C03638=1029.081,200.605,387.413,169.449,45.503,158.607
C03639=1029.086,200.854,387.389,169.452,45.500,158.607
C03640=1029.092,201.102,387.364,169.456,45.498,158.607
C03641=1029.098,201.351,387.340,169.460,45.496,158.607
C03642=1029.104,201.600,387.315,169.464,45.494,158.607
C03643=1029.110,201.849,387.290,169.468,45.491,158.607
C03644=1029.116,202.097,387.266,169.471,45.488,158.607
C03645=1029.122,202.346,387.240,169.474,45.486,158.607
C03646=1029.128,202.595,387.216,169.479,45.484,158.607
C03647=1029.134,202.843,387.191,169.482,45.482,158.607
C03648=1029.140,203.092,387.167,169.486,45.479,158.607
C03649=1029.146,203.341,387.142,169.490,45.477,158.606
C03650=1029.151,203.589,387.117,169.494,45.475,158.606
C03651=1029.157,203.839,387.092,169.498,45.472,158.606
C03652=1029.182,204.885,386.988,169.864,45.576,158.667
C03653=1029.194,205.258,386.949,169.867,45.574,158.667
C03654=1029.203,205.632,386.909,169.872,45.571,158.667
C03655=1029.213,206.005,386.870,169.876,45.569,158.667
C03656=1029.223,206.378,386.831,169.880,45.566,158.667
C03657=1029.230,206.628,386.805,169.883,45.565,158.667
C03658=1029.236,206.876,386.779,169.886,45.564,158.667
C03659=1029.243,207.124,386.752,169.889,45.562,158.667
C03660=1029.250,207.372,386.726,169.892,45.560,158.667
C03661=1029.256,207.621,386.699,169.895,45.559,158.667
C03662=1029.263,207.870,386.673,169.897,45.557,158.667
C03663=1029.270,208.118,386.647,169.900,45.556,158.667
C03664=1029.277,208.367,386.620,169.903,45.554,158.667
C03665=1029.284,208.615,386.594,169.905,45.553,158.667
C03666=1029.290,208.864,386.567,169.908,45.551,158.667
C03667=1029.297,209.112,386.541,169.911,45.550,158.667
C03668=1029.304,209.361,386.515,169.914,45.549,158.667
C03669=1029.309,209.609,386.488,169.916,45.547,158.666
C03670=1029.317,209.858,386.462,169.919,45.545,158.666
C03671=1029.324,210.107,386.435,169.923,45.544,158.666
C03672=1029.330,210.355,386.409,169.926,45.542,158.666
C03673=1029.337,210.604,386.382,169.928,45.541,158.667
C03674=1029.343,210.852,386.356,169.931,45.540,158.667
C03675=1029.350,211.101,386.330,169.934,45.538,158.666
C03676=1029.356,211.349,386.303,169.936,45.536,158.666
C03677=1029.363,211.598,386.277,169.939,45.535,158.666
C03678=1029.370,211.846,386.249,169.942,45.534,158.666
C03679=1029.376,212.094,386.223,169.945,45.532,158.666
C03680=1029.383,212.343,386.196,169.948,45.531,158.666
C03681=1029.389,212.591,386.170,169.950,45.530,158.666
C03682=1029.396,212.840,386.144,169.954,45.528,158.666
C03683=1029.403,213.089,386.117,169.957,45.527,158.667
C03684=1029.409,213.337,386.090,169.960,45.525,158.667
C03685=1029.416,213.586,386.063,169.962,45.524,158.667
C03686=1029.422,213.834,386.037,169.965,45.523,158.667
C03687=1029.429,214.083,386.010,169.968,45.521,158.667
C03688=1029.436,214.331,385.983,169.970,45.519,158.666
C03689=1029.442,214.579,385.956,169.973,45.518,158.666
C03690=1029.449,214.828,385.929,169.976,45.517,158.666
C03691=1029.456,215.077,385.903,169.979,45.515,158.666
C03692=1029.462,215.325,385.876,169.983,45.514,158.666
C03693=1029.469,215.573,385.849,169.985,45.512,158.666
C03694=1029.476,215.822,385.822,169.988,45.511,158.667
C03695=1029.482,216.070,385.796,169.991,45.510,158.667
C03696=1029.489,216.319,385.768,169.994,45.508,158.667
C03697=1029.496,216.568,385.742,169.996,45.507,158.667
C03698=1029.502,216.816,385.715,169.999,45.506,158.667
C03699=1029.509,217.064,385.688,170.002,45.504,158.667
C03700=1029.516,217.313,385.661,170.006,45.503,158.667
C03701=1029.523,217.562,385.635,170.009,45.501,158.667
C03702=1029.529,217.810,385.607,170.011,45.500,158.667
C03703=1029.536,218.058,385.581,170.014,45.499,158.667
C03704=1029.543,218.307,385.553,170.017,45.497,158.667
C03705=1029.549,218.555,385.527,170.020,45.496,158.667
C03706=1029.556,218.804,385.501,170.023,45.495,158.667
C03707=1029.563,219.052,385.473,170.026,45.493,158.667
C03708=1029.570,219.301,385.447,170.029,45.492,158.667
C03709=1029.579,219.679,385.406,170.034,45.490,158.667
C03710=1029.589,220.058,385.364,170.037,45.488,158.667
C03711=1029.599,220.437,385.322,170.042,45.486,158.667
C03712=1029.609,220.816,385.281,170.047,45.484,158.667
C03713=1029.616,221.065,385.254,170.050,45.483,158.667
C03714=1029.623,221.313,385.227,170.052,45.482,158.667
C03715=1029.630,221.562,385.200,170.055,45.480,158.667
C03716=1029.636,221.810,385.172,170.058,45.479,158.667
C03717=1029.642,222.059,385.145,170.062,45.477,158.667
C03718=1029.649,222.307,385.118,170.064,45.476,158.667
C03719=1029.656,222.556,385.090,170.068,45.475,158.667
C03720=1029.662,222.804,385.064,170.070,45.474,158.667
C03721=1029.669,223.053,385.036,170.073,45.473,158.667
C03722=1029.676,223.301,385.009,170.076,45.471,158.667
C03723=1029.682,223.550,384.982,170.079,45.470,158.667
C03724=1029.689,223.798,384.954,170.082,45.468,158.667
C03725=1029.695,224.046,384.927,170.085,45.467,158.667
C03726=1029.701,224.295,384.900,170.088,45.466,158.668
C03727=1029.709,224.543,384.873,170.091,45.465,158.668
C03728=1029.716,224.792,384.845,170.094,45.464,158.668
C03729=1029.722,225.041,384.818,170.098,45.462,158.668
C03730=1029.729,225.289,384.790,170.100,45.461,158.668
C03731=1029.735,225.537,384.763,170.103,45.460,158.668
C03732=1029.742,225.785,384.736,170.106,45.459,158.668
C03733=1029.749,226.034,384.709,170.109,45.457,158.668
C03734=1029.755,226.282,384.681,170.112,45.456,158.668
C03735=1029.763,226.531,384.654,170.115,45.454,158.668
C03736=1029.769,226.779,384.626,170.118,45.454,158.668
C03737=1029.776,227.027,384.598,170.121,45.452,158.668
C03738=1029.782,227.276,384.572,170.124,45.451,158.668
C03739=1029.789,227.524,384.545,170.127,45.450,158.668
C03740=1029.796,227.772,384.517,170.131,45.448,158.668
C03741=1029.803,228.021,384.489,170.134,45.447,158.668
C03742=1029.809,228.269,384.461,170.136,45.446,158.668
C03743=1029.816,228.518,384.434,170.139,45.445,158.668
C03744=1029.823,228.766,384.406,170.142,45.444,158.669
C03745=1029.829,229.015,384.378,170.146,45.443,158.669
C03746=1029.835,229.262,384.351,170.149,45.441,158.669
C03747=1029.842,229.511,384.324,170.152,45.440,158.669
C03748=1029.848,229.760,384.296,170.155,45.439,158.669
C03749=1029.855,230.008,384.268,170.157,45.438,158.669
C03750=1029.862,230.257,384.241,170.161,45.437,158.669
C03751=1029.868,230.505,384.213,170.164,45.436,158.669
C03752=1029.875,230.754,384.185,170.167,45.434,158.669
C03753=1029.882,231.002,384.157,170.170,45.433,158.669
C03754=1029.888,231.250,384.130,170.173,45.432,158.669
C03755=1029.895,231.499,384.101,170.176,45.431,158.669
C03756=1029.901,231.747,384.073,170.180,45.430,158.669
C03757=1029.908,231.995,384.045,170.182,45.429,158.669
C03758=1029.914,232.243,384.018,170.185,45.428,158.670
C03759=1029.921,232.492,383.990,170.188,45.427,158.670
C03760=1029.928,232.740,383.962,170.191,45.426,158.670
C03761=1029.933,232.989,383.934,170.195,45.424,158.670
C03762=1029.940,233.237,383.906,170.198,45.424,158.670
C03763=1029.947,233.485,383.878,170.201,45.422,158.670
C03764=1029.954,233.734,383.850,170.204,45.422,158.670
C03765=1029.964,234.105,383.808,170.209,45.420,158.670
C03766=1029.973,234.476,383.766,170.213,45.418,158.670
C03767=1029.984,234.848,383.725,170.218,45.416,158.671
C03768=1029.994,235.219,383.683,170.223,45.414,158.671
C03769=1030.000,235.467,383.655,170.226,45.414,158.671
C03770=1030.006,235.716,383.627,170.229,45.412,158.671
C03771=1030.013,235.964,383.599,170.232,45.412,158.671
C03772=1030.020,236.212,383.571,170.236,45.410,158.671
C03773=1030.026,236.460,383.543,170.239,45.409,158.671
C03774=1030.033,236.709,383.515,170.241,45.408,158.671
C03775=1030.040,236.958,383.487,170.244,45.407,158.671
C03776=1030.047,237.206,383.458,170.248,45.406,158.671
C03777=1030.053,237.455,383.430,170.251,45.405,158.672
C03778=1030.060,237.703,383.403,170.254,45.404,158.672
C03779=1030.067,237.951,383.374,170.257,45.403,158.672
C03780=1030.073,238.200,383.346,170.261,45.401,158.672
C03781=1030.080,238.448,383.318,170.264,45.401,158.672
C03782=1030.087,238.696,383.290,170.267,45.400,158.672
C03783=1030.093,238.944,383.262,170.270,45.399,158.672
C03784=1030.100,239.192,383.233,170.274,45.398,158.672
C03785=1030.106,239.441,383.205,170.277,45.396,158.672
C03786=1030.113,239.689,383.177,170.280,45.396,158.673
C03787=1030.120,239.937,383.149,170.282,45.394,158.673
C03788=1030.126,240.187,383.120,170.286,45.394,158.673
C03789=1030.133,240.434,383.092,170.289,45.393,158.673
C03790=1030.139,240.683,383.064,170.292,45.392,158.673
C03791=1030.146,240.931,383.035,170.295,45.391,158.673
C03792=1030.153,241.179,383.007,170.299,45.390,158.673
C03793=1030.159,241.428,382.978,170.302,45.389,158.673
C03794=1030.166,241.675,382.950,170.305,45.388,158.674
C03795=1030.172,241.924,382.922,170.309,45.387,158.674
C03796=1030.179,242.172,382.893,170.312,45.386,158.674
C03797=1030.186,242.421,382.864,170.315,45.385,158.674
C03798=1030.193,242.669,382.836,170.318,45.384,158.674
C03799=1030.199,242.917,382.807,170.322,45.383,158.674
C03800=1030.206,243.165,382.778,170.325,45.382,158.674
C03801=1030.212,243.414,382.750,170.328,45.381,158.675
C03802=1030.219,243.662,382.722,170.331,45.381,158.675
C03803=1030.225,243.910,382.693,170.335,45.380,158.675
C03804=1030.232,244.159,382.665,170.338,45.378,158.675
C03805=1030.239,244.407,382.636,170.341,45.378,158.675
C03806=1030.245,244.655,382.606,170.345,45.377,158.675
C03807=1030.251,244.903,382.577,170.348,45.376,158.675
C03808=1030.258,245.152,382.550,170.351,45.375,158.676
C03809=1030.264,245.400,382.521,170.354,45.375,158.676
C03810=1030.270,245.648,382.492,170.358,45.373,158.676
C03811=1030.277,245.897,382.462,170.361,45.372,158.676
C03812=1030.284,246.145,382.434,170.364,45.372,158.676
C03813=1030.290,246.393,382.405,170.367,45.371,158.676
C03814=1030.297,246.641,382.376,170.371,45.370,158.677
C03815=1030.303,246.890,382.347,170.374,45.369,158.677
C03816=1030.310,247.138,382.319,170.377,45.369,158.677
C03817=1030.317,247.386,382.290,170.380,45.368,158.677
C03818=1030.323,247.635,382.260,170.384,45.367,158.677
C03819=1030.329,247.883,382.231,170.387,45.366,158.677
C03820=1030.335,248.131,382.202,170.390,45.365,158.678
C03821=1030.346,248.497,382.160,170.395,45.364,158.678
C03822=1030.355,248.861,382.117,170.400,45.363,158.678
C03823=1030.365,249.227,382.074,170.405,45.362,158.678
C03824=1030.374,249.592,382.032,170.410,45.360,158.679
C03825=1030.381,249.840,382.003,170.413,45.360,158.679
C03826=1030.387,250.089,381.973,170.416,45.359,158.679
C03827=1030.394,250.337,381.945,170.420,45.358,158.679
C03828=1030.401,250.585,381.916,170.423,45.357,158.679
C03829=1030.407,250.834,381.887,170.426,45.357,158.680
C03830=1030.414,251.082,381.858,170.430,45.356,158.680
C03831=1030.420,251.330,381.828,170.433,45.355,158.680
C03832=1030.427,251.577,381.799,170.436,45.354,158.680
C03833=1030.434,251.826,381.770,170.440,45.353,158.680
C03834=1030.440,252.074,381.741,170.443,45.353,158.680
C03835=1030.447,252.323,381.712,170.446,45.352,158.681
C03836=1030.453,252.571,381.682,170.451,45.351,158.681
C03837=1030.460,252.819,381.654,170.454,45.350,158.681
C03838=1030.467,253.067,381.625,170.457,45.349,158.681
C03839=1030.474,253.316,381.595,170.461,45.349,158.681
C03840=1030.480,253.564,381.566,170.464,45.348,158.682
C03841=1030.487,253.813,381.536,170.468,45.347,158.682
C03842=1030.494,254.060,381.508,170.471,45.347,158.682
C03843=1030.500,254.308,381.479,170.474,45.346,158.682
C03844=1030.507,254.557,381.449,170.478,45.345,158.682
C03845=1030.514,254.805,381.420,170.481,45.344,158.682
C03846=1030.520,255.054,381.390,170.485,45.343,158.683
C03847=1030.527,255.301,381.362,170.488,45.343,158.683
C03848=1030.534,255.549,381.332,170.491,45.342,158.683
C03849=1030.541,255.798,381.303,170.495,45.341,158.683
C03850=1030.547,256.046,381.274,170.498,45.340,158.683
C03851=1030.554,256.294,381.244,170.502,45.339,158.684
C03852=1030.560,256.542,381.215,170.505,45.339,158.684
C03853=1030.568,256.791,381.186,170.508,45.338,158.684
C03854=1030.575,257.038,381.156,170.512,45.337,158.684
C03855=1030.581,257.287,381.127,170.515,45.336,158.684
C03856=1030.588,257.535,381.097,170.519,45.335,158.685
C03857=1030.594,257.783,381.068,170.522,45.335,158.685
C03858=1030.602,258.031,381.039,170.525,45.334,158.685
C03859=1030.608,258.279,381.010,170.529,45.333,158.685
C03860=1030.615,258.528,380.980,170.533,45.333,158.685
C03861=1030.622,258.776,380.951,170.537,45.332,158.686
C03862=1030.629,259.024,380.921,170.540,45.331,158.686
C03863=1030.636,259.273,380.891,170.544,45.331,158.686
C03864=1030.643,259.520,380.862,170.547,45.330,158.686
C03865=1030.650,259.769,380.833,170.551,45.329,158.686
C03866=1030.656,260.017,380.804,170.554,45.328,158.687
C03867=1030.663,260.265,380.773,170.558,45.327,158.687
C03868=1030.669,260.513,380.744,170.561,45.327,158.687
C03869=1030.676,260.762,380.714,170.564,45.327,158.687
C03870=1030.684,261.009,380.685,170.568,45.326,158.688
C03871=1030.691,261.258,380.656,170.571,45.325,158.688
C03872=1030.696,261.505,380.625,170.575,45.324,158.688
C03873=1030.703,261.754,380.596,170.579,45.324,158.688
C03874=1030.710,262.002,380.566,170.583,45.323,158.688
C03875=1030.717,262.250,380.536,170.586,45.322,158.689
C03876=1030.724,262.497,380.506,170.589,45.322,158.689
C03877=1030.733,262.862,380.462,170.594,45.321,158.689
C03878=1030.743,263.226,380.418,170.600,45.320,158.690
C03879=1030.752,263.590,380.374,170.606,45.319,158.690
C03880=1030.762,263.954,380.330,170.611,45.319,158.690
C03881=1030.769,264.202,380.300,170.614,45.318,158.691
C03882=1030.775,264.450,380.271,170.618,45.317,158.691
C03883=1030.783,264.698,380.241,170.621,45.317,158.691
C03884=1030.789,264.947,380.210,170.624,45.316,158.691
C03885=1030.796,265.194,380.181,170.629,45.316,158.692
C03886=1030.803,265.442,380.150,170.632,45.315,158.692
C03887=1030.809,265.690,380.121,170.636,45.314,158.692
C03888=1030.816,265.938,380.090,170.639,45.314,158.692
C03889=1030.823,266.187,380.061,170.643,45.313,158.693
C03890=1030.829,266.435,380.031,170.646,45.313,158.693
C03891=1030.836,266.683,380.001,170.650,45.312,158.693
C03892=1030.843,266.932,379.970,170.654,45.312,158.694
C03893=1030.849,267.179,379.940,170.658,45.311,158.694
C03894=1030.856,267.427,379.910,170.661,45.311,158.694
C03895=1030.863,267.676,379.879,170.665,45.310,158.694
C03896=1030.869,267.923,379.850,170.668,45.310,158.695
C03897=1030.876,268.172,379.819,170.672,45.309,158.695
C03898=1030.883,268.420,379.789,170.676,45.309,158.695
C03899=1030.890,268.667,379.758,170.680,45.308,158.695
C03900=1030.896,268.915,379.728,170.683,45.308,158.696
C03901=1030.903,269.164,379.698,170.687,45.307,158.696
C03902=1030.909,269.411,379.667,170.690,45.307,158.696
C03903=1030.916,269.660,379.637,170.694,45.306,158.696
C03904=1030.924,269.908,379.607,170.698,45.306,158.697
C03905=1030.929,270.156,379.577,170.702,45.306,158.697
C03906=1030.937,270.404,379.546,170.705,45.305,158.697
C03907=1030.943,270.652,379.515,170.709,45.305,158.698
C03908=1030.950,270.900,379.485,170.712,45.304,158.698
C03909=1030.956,271.148,379.455,170.717,45.304,158.698
C03910=1030.963,271.396,379.424,170.720,45.304,158.699
C03911=1030.970,271.644,379.393,170.724,45.303,158.699
C03912=1030.977,271.892,379.363,170.727,45.303,158.699
C03913=1030.983,272.140,379.333,170.732,45.303,158.700
C03914=1030.989,272.389,379.302,170.735,45.302,158.700
C03915=1030.997,272.636,379.271,170.739,45.302,158.700
C03916=1031.003,272.885,379.240,170.742,45.302,158.700
C03917=1031.010,273.132,379.210,170.746,45.301,158.701
C03918=1031.017,273.380,379.179,170.750,45.301,158.701
C03919=1031.024,273.628,379.149,170.754,45.300,158.701
C03920=1031.031,273.876,379.118,170.757,45.300,158.702
C03921=1031.036,274.124,379.087,170.761,45.300,158.702
C03922=1031.043,274.372,379.057,170.764,45.299,158.702
C03923=1031.050,274.620,379.026,170.769,45.299,158.703
C03924=1031.057,274.869,378.995,170.772,45.299,158.703
C03925=1031.064,275.116,378.964,170.776,45.298,158.703
C03926=1031.071,275.365,378.933,170.780,45.298,158.704
C03927=1031.077,275.612,378.902,170.784,45.298,158.704
C03928=1031.084,275.860,378.872,170.788,45.298,158.704
C03929=1031.091,276.108,378.841,170.791,45.297,158.705
C03930=1031.097,276.357,378.810,170.795,45.297,158.705
C03931=1031.104,276.604,378.779,170.799,45.296,158.705
C03932=1031.111,276.853,378.748,170.803,45.296,158.705
C03933=1031.121,277.221,378.702,170.808,45.296,158.706
C03934=1031.131,277.589,378.657,170.815,45.295,158.706
C03935=1031.141,277.957,378.610,170.820,45.295,158.707
C03936=1031.151,278.327,378.564,170.826,45.294,158.707
C03937=1031.157,278.574,378.533,170.830,45.294,158.708
C03938=1031.164,278.822,378.502,170.833,45.294,158.708
C03939=1031.171,279.070,378.471,170.837,45.294,158.709
C03940=1031.177,279.319,378.440,170.841,45.294,158.709
C03941=1031.184,279.566,378.408,170.845,45.293,158.709
C03942=1031.191,279.814,378.377,170.849,45.293,158.710
C03943=1031.197,280.062,378.346,170.853,45.293,158.710
C03944=1031.204,280.310,378.314,170.857,45.293,158.710
C03945=1031.211,280.559,378.283,170.860,45.293,158.711
C03946=1031.218,280.806,378.253,170.865,45.292,158.711
C03947=1031.225,281.054,378.221,170.869,45.292,158.711
C03948=1031.232,281.302,378.190,170.872,45.292,158.712
C03949=1031.238,281.550,378.158,170.876,45.292,158.712
C03950=1031.245,281.798,378.127,170.880,45.292,158.712
C03951=1031.252,282.046,378.095,170.884,45.291,158.713
C03952=1031.258,282.294,378.064,170.888,45.291,158.713
C03953=1031.265,282.542,378.032,170.892,45.291,158.714
C03954=1031.272,282.790,378.002,170.896,45.291,158.714
C03955=1031.278,283.038,377.970,170.900,45.290,158.714
C03956=1031.285,283.286,377.939,170.904,45.290,158.715
C03957=1031.292,283.534,377.907,170.908,45.290,158.715
C03958=1031.299,283.781,377.877,170.912,45.290,158.716
C03959=1031.306,284.029,377.845,170.916,45.290,158.716
C03960=1031.313,284.277,377.814,170.920,45.290,158.716
C03961=1031.319,284.525,377.782,170.923,45.290,158.717
C03962=1031.326,284.772,377.750,170.928,45.290,158.717
C03963=1031.333,285.020,377.719,170.932,45.289,158.717
C03964=1031.340,285.268,377.687,170.935,45.289,158.718
C03965=1031.347,285.516,377.656,170.940,45.289,158.718
C03966=1031.353,285.764,377.624,170.944,45.289,158.719
C03967=1031.360,286.012,377.593,170.948,45.289,158.719
C03968=1031.367,286.260,377.562,170.952,45.289,158.719
C03969=1031.374,286.508,377.530,170.956,45.289,158.720
C03970=1031.381,286.756,377.498,170.960,45.288,158.720
C03971=1031.388,287.004,377.466,170.964,45.289,158.721
C03972=1031.395,287.251,377.435,170.968,45.289,158.721
C03973=1031.401,287.500,377.403,170.972,45.288,158.721
C03974=1031.408,287.747,377.371,170.976,45.289,158.722
C03975=1031.414,287.995,377.339,170.980,45.289,158.722
C03976=1031.421,288.243,377.308,170.985,45.288,158.723
C03977=1031.429,288.491,377.275,170.988,45.288,158.723
C03978=1031.435,288.739,377.244,170.992,45.289,158.723
C03979=1031.442,288.987,377.212,170.997,45.288,158.724
C03980=1031.448,289.234,377.180,171.000,45.288,158.724
C03981=1031.455,289.482,377.148,171.005,45.288,158.725
C03982=1031.462,289.729,377.116,171.009,45.288,158.725
C03983=1031.469,289.978,377.084,171.013,45.289,158.726
C03984=1031.476,290.226,377.052,171.017,45.288,158.726
C03985=1031.482,290.473,377.020,171.021,45.288,158.726
C03986=1031.489,290.721,376.989,171.026,45.288,158.727
C03987=1031.496,290.969,376.956,171.029,45.288,158.727
C03988=1031.503,291.218,376.924,171.034,45.289,158.728
C03989=1031.514,291.598,376.875,171.040,45.289,158.728
C03990=1031.524,291.978,376.826,171.047,45.288,158.729
C03991=1031.535,292.359,376.776,171.052,45.289,158.730
C03992=1031.546,292.739,376.727,171.059,45.288,158.730
C03993=1031.552,292.987,376.695,171.063,45.289,158.731
C03994=1031.559,293.236,376.663,171.067,45.289,158.731
C03995=1031.566,293.483,376.630,171.071,45.289,158.732
C03996=1031.573,293.731,376.598,171.076,45.289,158.732
C03997=1031.579,293.978,376.566,171.080,45.289,158.733
C03998=1031.586,294.227,376.533,171.084,45.290,158.733
C03999=1031.593,294.474,376.501,171.088,45.289,158.734
C04000=1031.599,294.722,376.468,171.093,45.290,158.734
C04001=1031.606,294.969,376.437,171.097,45.290,158.735
C04002=1031.613,295.218,376.404,171.100,45.290,158.735
C04003=1031.619,295.465,376.371,171.105,45.290,158.735
C04004=1031.626,295.713,376.339,171.110,45.290,158.736
C04005=1031.633,295.961,376.306,171.114,45.290,158.736
C04006=1031.640,296.209,376.273,171.117,45.291,158.737
C04007=1031.647,296.456,376.241,171.122,45.291,158.737
C04008=1031.653,296.703,376.208,171.127,45.291,158.738
C04009=1031.660,296.952,376.175,171.131,45.292,158.739
C04010=1031.667,297.199,376.143,171.134,45.292,158.739
C04011=1031.673,297.447,376.110,171.139,45.292,158.739
C04012=1031.680,297.695,376.077,171.144,45.292,158.740
C04013=1031.686,297.942,376.044,171.148,45.293,158.741
C04014=1031.694,298.190,376.012,171.151,45.292,158.741
C04015=1031.700,298.438,375.979,171.156,45.293,158.741
C04016=1031.707,298.686,375.946,171.161,45.293,158.742
C04017=1031.714,298.934,375.914,171.165,45.293,158.742
C04018=1031.721,299.181,375.880,171.170,45.294,158.743
C04019=1031.728,299.429,375.847,171.173,45.294,158.744
C04020=1031.734,299.676,375.815,171.178,45.294,158.744
C04021=1031.741,299.924,375.782,171.182,45.294,158.744
C04022=1031.748,300.172,375.749,171.187,45.295,158.745
C04023=1031.754,300.420,375.717,171.191,45.295,158.746
C04024=1031.762,300.667,375.683,171.196,45.295,158.746
C04025=1031.768,300.915,375.651,171.199,45.296,158.747
C04026=1031.775,301.163,375.617,171.204,45.296,158.747
C04027=1031.782,301.411,375.585,171.209,45.296,158.748
C04028=1031.790,301.658,375.552,171.213,45.297,158.748
C04029=1031.796,301.905,375.519,171.218,45.297,158.749
C04030=1031.803,302.154,375.486,171.222,45.297,158.749
C04031=1031.810,302.400,375.453,171.226,45.298,158.750
C04032=1031.817,302.649,375.420,171.230,45.298,158.750
C04033=1031.823,302.896,375.387,171.235,45.298,158.751
C04034=1031.830,303.144,375.353,171.239,45.298,158.751
C04035=1031.837,303.391,375.321,171.244,45.298,158.752
C04036=1031.844,303.640,375.288,171.248,45.299,158.752
C04037=1031.851,303.887,375.254,171.253,45.299,158.753
C04038=1031.858,304.135,375.221,171.258,45.299,158.753
C04039=1031.866,304.382,375.188,171.261,45.300,158.754
C04040=1031.872,304.630,375.155,171.266,45.300,158.755
C04041=1031.879,304.877,375.121,171.270,45.301,158.755
C04042=1031.886,305.125,375.089,171.275,45.302,158.756
C04043=1031.894,305.372,375.056,171.280,45.302,158.756
C04044=1031.900,305.621,375.022,171.284,45.302,158.757
C04045=1031.911,306.018,374.969,171.291,45.303,158.758
C04046=1031.922,306.416,374.916,171.299,45.303,158.759
C04047=1031.934,306.814,374.863,171.306,45.304,158.760
C04048=1031.945,307.211,374.809,171.313,45.304,158.760
C04049=1031.952,307.459,374.776,171.317,45.305,158.761
C04050=1031.960,307.706,374.742,171.322,45.306,158.762
C04051=1031.967,307.953,374.709,171.327,45.306,158.762
C04052=1031.974,308.202,374.676,171.331,45.306,158.763
C04053=1031.981,308.449,374.642,171.336,45.307,158.763
C04054=1031.989,308.697,374.609,171.341,45.307,158.764
C04055=1031.995,308.944,374.576,171.345,45.307,158.764
C04056=1032.002,309.192,374.542,171.350,45.308,158.765
C04057=1032.010,309.440,374.508,171.355,45.308,158.766
C04058=1032.017,309.687,374.474,171.359,45.309,158.766
C04059=1032.024,309.935,374.442,171.364,45.309,158.767
C04060=1032.031,310.182,374.409,171.368,45.310,158.767
C04061=1032.038,310.430,374.375,171.373,45.310,158.768
C04062=1032.045,310.678,374.341,171.378,45.311,158.769
C04063=1032.053,310.925,374.308,171.382,45.311,158.769
C04064=1032.060,311.173,374.275,171.387,45.312,158.770
C04065=1032.067,311.421,374.241,171.392,45.312,158.770
C04066=1032.074,311.668,374.206,171.396,45.312,158.771
C04067=1032.081,311.915,374.172,171.401,45.313,158.772
C04068=1032.088,312.163,374.138,171.406,45.314,158.772
C04069=1032.094,312.411,374.104,171.410,45.315,158.773
C04070=1032.101,312.658,374.070,171.415,45.315,158.774
C04071=1032.108,312.906,374.037,171.420,45.316,158.774
C04072=1032.115,313.154,374.002,171.425,45.317,158.775
C04073=1032.122,313.401,373.968,171.429,45.317,158.775
C04074=1032.129,313.648,373.934,171.434,45.318,158.776
C04075=1032.136,313.896,373.899,171.439,45.319,158.777
C04076=1032.142,314.143,373.866,171.443,45.319,158.777
C04077=1032.149,314.391,373.831,171.448,45.320,158.778
C04078=1032.156,314.638,373.797,171.453,45.321,158.779
C04079=1032.164,314.886,373.763,171.458,45.321,158.779
C04080=1032.170,315.134,373.729,171.462,45.322,158.780
C04081=1032.178,315.381,373.694,171.467,45.323,158.781
C04082=1032.184,315.629,373.660,171.472,45.323,158.781
C04083=1032.192,315.876,373.625,171.477,45.324,158.782
C04084=1032.199,316.124,373.591,171.482,45.325,158.783
C04085=1032.205,316.372,373.557,171.486,45.325,158.783
C04086=1032.212,316.618,373.523,171.491,45.326,158.784
C04087=1032.219,316.866,373.488,171.496,45.327,158.785
C04088=1032.226,317.113,373.454,171.501,45.328,158.785
C04089=1032.233,317.361,373.420,171.505,45.329,158.786
C04090=1032.240,317.609,373.386,171.510,45.329,158.787
C04091=1032.247,317.856,373.351,171.515,45.330,158.787
C04092=1032.254,318.104,373.317,171.520,45.331,158.788
C04093=1032.261,318.351,373.282,171.524,45.332,158.789
C04094=1032.269,318.599,373.247,171.529,45.332,158.789
C04095=1032.276,318.847,373.213,171.535,45.333,158.790
C04096=1032.283,319.094,373.178,171.540,45.334,158.791
C04097=1032.290,319.342,373.144,171.545,45.335,158.792
C04098=1032.297,319.589,373.109,171.549,45.336,158.792
C04099=1032.304,319.836,373.075,171.554,45.336,158.793
C04100=1032.311,320.084,373.040,171.559,45.337,158.794
C04101=1032.323,320.486,372.984,171.567,45.339,158.795
C04102=1032.334,320.888,372.927,171.575,45.340,158.796
C04103=1032.347,321.292,372.871,171.583,45.342,158.797
C04104=1032.358,321.694,372.815,171.591,45.342,158.798
C04105=1032.366,321.941,372.780,171.596,45.343,158.799
C04106=1032.372,322.189,372.745,171.601,45.344,158.800
C04107=1032.380,322.436,372.711,171.606,45.345,158.800
C04108=1032.387,322.684,372.676,171.612,45.346,158.801
C04109=1032.394,322.932,372.641,171.616,45.347,158.802
C04110=1032.401,323.179,372.606,171.621,45.348,158.803
C04111=1032.409,323.426,372.572,171.626,45.349,158.803
C04112=1032.417,323.674,372.537,171.631,45.349,158.804
C04113=1032.424,323.921,372.502,171.637,45.350,158.805
C04114=1032.431,324.168,372.467,171.642,45.351,158.805
C04115=1032.438,324.416,372.432,171.647,45.353,158.806
C04116=1032.446,324.663,372.397,171.651,45.353,158.807
C04117=1032.452,324.911,372.363,171.656,45.354,158.808
C04118=1032.460,325.159,372.328,171.662,45.355,158.809
C04119=1032.467,325.406,372.293,171.667,45.356,158.809
C04120=1032.475,325.653,372.258,171.672,45.357,158.810
C04121=1032.482,325.901,372.223,171.677,45.358,158.811
C04122=1032.490,326.148,372.187,171.682,45.358,158.811
C04123=1032.497,326.395,372.152,171.688,45.360,158.812
C04124=1032.505,326.643,372.117,171.692,45.361,158.813
C04125=1032.512,326.890,372.083,171.697,45.362,158.814
C04126=1032.520,327.138,372.047,171.703,45.362,158.815
C04127=1032.527,327.385,372.013,171.708,45.363,158.815
C04128=1032.534,327.633,371.978,171.713,45.365,158.816
C04129=1032.542,327.880,371.943,171.718,45.366,158.817
C04130=1032.549,328.127,371.907,171.724,45.366,158.818
C04131=1032.556,328.375,371.871,171.729,45.368,158.819
C04132=1032.563,328.622,371.836,171.734,45.369,158.819
C04133=1032.571,328.870,371.800,171.739,45.370,158.820
C04134=1032.578,329.117,371.765,171.745,45.371,158.821
C04135=1032.586,329.364,371.730,171.749,45.372,158.822
C04136=1032.593,329.612,371.694,171.755,45.373,158.823
C04137=1032.600,329.859,371.659,171.759,45.374,158.823
C04138=1032.607,330.107,371.623,171.766,45.375,158.824
C04139=1032.614,330.354,371.588,171.770,45.376,158.825
C04140=1032.622,330.601,371.551,171.775,45.378,158.826
C04141=1032.629,330.849,371.516,171.782,45.379,158.827
C04142=1032.636,331.096,371.480,171.786,45.380,158.827
C04143=1032.643,331.343,371.444,171.792,45.382,158.828
C04144=1032.651,331.591,371.409,171.797,45.382,158.829
C04145=1032.658,331.837,371.373,171.802,45.384,158.830
C04146=1032.666,332.086,371.338,171.807,45.385,158.831
C04147=1032.673,332.332,371.302,171.813,45.386,158.832
C04148=1032.681,332.580,371.266,171.819,45.387,158.833
C04149=1032.688,332.828,371.230,171.823,45.388,158.833
C04150=1032.695,333.075,371.195,171.829,45.389,158.834
C04151=1032.703,333.322,371.158,171.835,45.391,158.835
C04152=1032.710,333.569,371.122,171.839,45.392,158.836
C04153=1032.717,333.817,371.087,171.846,45.393,158.837
C04154=1032.725,334.064,371.051,171.851,45.395,158.838
C04155=1032.732,334.311,371.015,171.856,45.396,158.839
C04156=1032.740,334.558,370.979,171.862,45.397,158.839
C04157=1032.752,334.957,370.921,171.871,45.399,158.841
C04158=1032.764,335.355,370.862,171.879,45.401,158.842
C04159=1032.775,335.753,370.805,171.888,45.403,158.844
C04160=1032.787,336.151,370.746,171.897,45.405,158.845
C04161=1032.795,336.398,370.710,171.902,45.407,158.846
C04162=1032.802,336.645,370.674,171.908,45.408,158.847
C04163=1032.810,336.892,370.638,171.913,45.410,158.848
C04164=1032.816,337.140,370.601,171.918,45.411,158.849
C04165=1032.824,337.387,370.565,171.924,45.412,158.850
C04166=1032.831,337.634,370.529,171.929,45.414,158.851
C04167=1032.839,337.882,370.493,171.935,45.415,158.851
C04168=1032.847,338.128,370.456,171.940,45.417,158.852
C04169=1032.855,338.376,370.419,171.947,45.418,158.853
C04170=1032.861,338.624,370.383,171.952,45.419,158.854
C04171=1032.869,338.870,370.347,171.958,45.421,158.855
C04172=1032.876,339.118,370.311,171.963,45.422,158.856
C04173=1032.884,339.365,370.274,171.968,45.424,158.857
C04174=1032.892,339.612,370.237,171.974,45.425,158.858
C04175=1032.899,339.860,370.201,171.980,45.427,158.859
C04176=1032.907,340.107,370.164,171.986,45.428,158.860
C04177=1032.914,340.354,370.127,171.991,45.430,158.861
C04178=1032.922,340.602,370.091,171.997,45.431,158.862
C04179=1032.930,340.848,370.055,172.002,45.432,158.863
C04180=1032.936,341.095,370.018,172.008,45.434,158.864
C04181=1032.944,341.342,369.981,172.013,45.436,158.865
C04182=1032.951,341.590,369.944,172.020,45.437,158.866
C04183=1032.959,341.837,369.907,172.025,45.439,158.867
C04184=1032.967,342.084,369.871,172.031,45.440,158.868
C04185=1032.974,342.331,369.833,172.036,45.442,158.868
C04186=1032.982,342.578,369.797,172.043,45.444,158.870
C04187=1032.989,342.826,369.760,172.048,45.445,158.870
C04188=1032.997,343.073,369.723,172.054,45.446,158.871
C04189=1033.004,343.321,369.686,172.060,45.448,158.873
C04190=1033.012,343.567,369.649,172.065,45.450,158.873
C04191=1033.019,343.815,369.612,172.072,45.451,158.875
C04192=1033.027,344.061,369.575,172.077,45.453,158.875
C04193=1033.035,344.309,369.538,172.083,45.455,158.877
C04194=1033.042,344.556,369.501,172.088,45.456,158.877
C04195=1033.050,344.803,369.464,172.095,45.458,158.879
C04196=1033.057,345.050,369.426,172.100,45.460,158.879
C04197=1033.065,345.297,369.389,172.106,45.461,158.881
C04198=1033.072,345.544,369.353,172.112,45.463,158.882
C04199=1033.080,345.792,369.315,172.118,45.465,158.883
C04200=1033.088,346.038,369.278,172.124,45.466,158.884
C04201=1033.095,346.286,369.241,172.129,45.468,158.885
C04202=1033.103,346.533,369.203,172.136,45.470,158.886
C04203=1033.111,346.780,369.166,172.142,45.471,158.887
C04204=1033.119,347.027,369.129,172.147,45.473,158.888
C04205=1033.126,347.274,369.091,172.154,45.475,158.889
C04206=1033.134,347.521,369.054,172.160,45.477,158.890
C04207=1033.141,347.768,369.017,172.165,45.478,158.891
C04208=1033.150,348.016,368.980,172.171,45.480,158.892
C04209=1033.157,348.263,368.942,172.178,45.482,158.893
C04210=1033.165,348.509,368.904,172.183,45.484,158.894
C04211=1033.173,348.756,368.867,172.189,45.485,158.895
C04212=1033.180,349.003,368.829,172.196,45.487,158.896
C04213=1033.193,349.398,368.769,172.205,45.490,158.898
C04214=1033.204,349.793,368.709,172.215,45.493,158.900
C04215=1033.217,350.188,368.649,172.224,45.496,158.902
C04216=1033.230,350.582,368.588,172.235,45.499,158.903
C04217=1033.237,350.829,368.551,172.240,45.501,158.904
C04218=1033.245,351.077,368.512,172.247,45.503,158.906
C04219=1033.252,351.324,368.475,172.253,45.505,158.907
C04220=1033.260,351.571,368.437,172.258,45.507,158.908
C04221=1033.268,351.818,368.399,172.265,45.509,158.909
C04222=1033.276,352.064,368.361,172.271,45.511,158.910
C04223=1033.283,352.311,368.323,172.277,45.512,158.911
C04224=1033.291,352.559,368.285,172.283,45.514,158.912
C04225=1033.299,352.806,368.247,172.289,45.516,158.913
C04226=1033.307,353.053,368.209,172.296,45.519,158.915
C04227=1033.315,353.300,368.172,172.302,45.520,158.916
C04228=1033.322,353.546,368.134,172.308,45.522,158.917
C04229=1033.330,353.793,368.095,172.314,45.524,158.918
C04230=1033.338,354.041,368.057,172.321,45.526,158.919
C04231=1033.346,354.288,368.019,172.327,45.529,158.920
C04232=1033.354,354.534,367.981,172.334,45.530,158.921
C04233=1033.362,354.781,367.943,172.340,45.532,158.923
C04234=1033.369,355.028,367.905,172.346,45.535,158.924
C04235=1033.378,355.276,367.866,172.352,45.537,158.925
C04236=1033.385,355.522,367.828,172.359,45.538,158.926
C04237=1033.393,355.769,367.790,172.365,45.541,158.927
C04238=1033.401,356.016,367.751,172.372,45.543,158.929
C04239=1033.409,356.263,367.713,172.378,45.545,158.930
C04240=1033.417,356.510,367.674,172.384,45.547,158.931
C04241=1033.425,356.757,367.636,172.390,45.549,158.932
C04242=1033.433,357.004,367.597,172.397,45.551,158.933
C04243=1033.440,357.251,367.559,172.403,45.554,158.935
C04244=1033.449,357.498,367.520,172.410,45.555,158.936
C04245=1033.456,357.744,367.482,172.417,45.558,158.937
C04246=1033.464,357.991,367.444,172.423,45.560,158.938
C04247=1033.472,358.239,367.405,172.430,45.562,158.939
C04248=1033.480,358.485,367.366,172.435,45.564,158.941
C04249=1033.488,358.732,367.327,172.442,45.566,158.942
C04250=1033.497,358.979,367.289,172.448,45.569,158.943
C04251=1033.504,359.226,367.250,172.455,45.571,158.944
C04252=1033.513,359.472,367.211,172.461,45.573,158.946
C04253=1033.521,359.719,367.173,172.468,45.575,158.947
C04254=1033.529,359.967,367.134,172.475,45.578,158.948
C04255=1033.537,360.212,367.095,172.481,45.580,158.949
C04256=1033.545,360.460,367.056,172.488,45.582,158.951
C04257=1033.552,360.707,367.017,172.495,45.584,158.952
C04258=1033.561,360.954,366.978,172.501,45.587,158.953
C04259=1033.568,361.200,366.940,172.508,45.589,158.955
C04260=1033.577,361.447,366.900,172.515,45.591,158.956
C04261=1033.585,361.694,366.862,172.521,45.594,158.957
C04262=1033.593,361.941,366.822,172.528,45.596,158.958
C04263=1033.601,362.188,366.782,172.535,45.599,158.960
C04264=1033.609,362.434,366.744,172.541,45.601,158.961
C04265=1033.616,362.681,366.704,172.548,45.603,158.962
C04266=1033.625,362.928,366.665,172.555,45.606,158.964
C04267=1033.633,363.175,366.626,172.561,45.608,158.965
C04268=1033.641,363.422,366.586,172.568,45.610,158.966
C04269=1033.653,363.822,366.523,172.579,45.615,158.968
C04270=1033.667,364.224,366.459,172.590,45.619,158.971
C04271=1033.680,364.624,366.394,172.602,45.622,158.973
C04272=1033.693,365.025,366.331,172.612,45.626,158.975
C04273=1033.701,365.272,366.291,172.619,45.629,158.976
C04274=1033.710,365.518,366.252,172.626,45.632,158.978
C04275=1033.717,365.765,366.212,172.633,45.634,158.979
C04276=1033.726,366.012,366.173,172.640,45.637,158.981
C04277=1033.734,366.258,366.133,172.647,45.639,158.982
C04278=1033.742,366.505,366.093,172.654,45.641,158.983
C04279=1033.751,366.752,366.054,172.661,45.644,158.985
C04280=1033.759,366.999,366.014,172.668,45.647,158.986
C04281=1033.767,367.246,365.975,172.675,45.650,158.988
C04282=1033.776,367.492,365.934,172.681,45.652,158.989
C04283=1033.784,367.739,365.895,172.689,45.654,158.990
C04284=1033.792,367.985,365.855,172.696,45.657,158.992
C04285=1033.801,368.232,365.816,172.703,45.659,158.993
C04286=1033.808,368.479,365.776,172.710,45.662,158.995
C04287=1033.817,368.725,365.736,172.717,45.665,158.996
C04288=1033.825,368.972,365.696,172.724,45.667,158.997
C04289=1033.834,369.219,365.656,172.731,45.670,158.999
C04290=1033.843,369.465,365.616,172.738,45.673,159.000
C04291=1033.850,369.712,365.576,172.745,45.676,159.002
C04292=1033.859,369.959,365.535,172.753,45.678,159.003
C04293=1033.867,370.206,365.496,172.760,45.681,159.005
C04294=1033.875,370.452,365.455,172.767,45.684,159.006
C04295=1033.883,370.699,365.415,172.774,45.687,159.008
C04296=1033.892,370.945,365.375,172.782,45.689,159.009
C04297=1033.901,371.192,365.334,172.789,45.692,159.011
C04298=1033.908,371.439,365.295,172.796,45.695,159.012
C04299=1033.917,371.685,365.254,172.804,45.698,159.014
C04300=1033.925,371.931,365.214,172.811,45.701,159.015
C04301=1033.934,372.178,365.173,172.818,45.704,159.017
C04302=1033.941,372.425,365.133,172.825,45.707,159.018
C04303=1033.950,372.671,365.093,172.833,45.709,159.020
C04304=1033.959,372.918,365.052,172.840,45.712,159.021
C04305=1033.967,373.164,365.011,172.847,45.715,159.023
C04306=1033.975,373.410,364.971,172.855,45.718,159.024
C04307=1033.984,373.657,364.930,172.862,45.721,159.026
C04308=1033.992,373.903,364.890,172.870,45.724,159.027
C04309=1034.001,374.150,364.849,172.877,45.727,159.029
C04310=1034.010,374.396,364.809,172.884,45.730,159.030
C04311=1034.018,374.642,364.768,172.892,45.733,159.032
C04312=1034.026,374.889,364.727,172.899,45.735,159.033
C04313=1034.034,375.136,364.686,172.907,45.739,159.035
C04314=1034.044,375.382,364.646,172.914,45.742,159.037
C04315=1034.052,375.629,364.605,172.921,45.745,159.038
C04316=1034.060,375.876,364.564,172.929,45.748,159.040
C04317=1034.069,376.123,364.523,172.936,45.751,159.041
C04318=1034.078,376.368,364.482,172.944,45.753,159.043
C04319=1034.087,376.615,364.441,172.952,45.757,159.045
C04320=1034.095,376.861,364.401,172.959,45.759,159.046
C04321=1034.103,377.108,364.360,172.967,45.763,159.048
C04322=1034.112,377.354,364.319,172.975,45.766,159.049
C04323=1034.121,377.601,364.278,172.982,45.769,159.051
C04324=1034.130,377.848,364.237,172.990,45.772,159.053
C04325=1034.137,378.058,364.201,172.997,45.775,159.054
C04326=1034.145,378.269,364.166,173.003,45.777,159.055
C04327=1034.152,378.480,364.131,173.010,45.780,159.057
C04328=1034.159,378.690,364.096,173.016,45.782,159.058
C04329=1034.166,378.901,364.060,173.023,45.785,159.060
C04330=1034.174,379.112,364.025,173.029,45.788,159.061
C04331=1034.181,379.323,363.990,173.036,45.791,159.062
C04332=1034.189,379.533,363.954,173.043,45.794,159.064
C04333=1034.197,379.780,363.913,173.050,45.797,159.066
C04334=1034.205,380.026,363.871,173.059,45.800,159.067
C04335=1034.214,380.273,363.829,173.067,45.804,159.069
C04336=1034.223,380.519,363.788,173.074,45.807,159.071
C04337=1034.231,380.766,363.747,173.083,45.810,159.073
C04338=1034.240,381.012,363.705,173.090,45.814,159.074
C04339=1034.249,381.258,363.663,173.098,45.817,159.076
C04340=1034.258,381.504,363.622,173.106,45.820,159.078
C04341=1034.267,381.751,363.580,173.114,45.824,159.079
C04342=1034.275,381.997,363.538,173.122,45.827,159.081
C04343=1034.284,382.243,363.497,173.130,45.830,159.083
C04344=1034.293,382.490,363.455,173.139,45.833,159.085
C04345=1034.301,382.736,363.413,173.146,45.837,159.086
C04346=1034.310,382.982,363.371,173.154,45.840,159.088
C04347=1034.319,383.229,363.330,173.162,45.843,159.090
C04348=1034.328,383.474,363.287,173.170,45.847,159.092
C04349=1034.337,383.721,363.245,173.178,45.850,159.093
C04350=1034.346,383.967,363.204,173.187,45.853,159.095
C04351=1034.355,384.213,363.162,173.195,45.857,159.097
C04352=1034.364,384.460,363.120,173.202,45.861,159.099
C04353=1034.373,384.705,363.078,173.211,45.864,159.100
C04354=1034.382,384.952,363.036,173.219,45.868,159.102
C04355=1034.390,385.199,362.994,173.228,45.871,159.104
C04356=1034.399,385.444,362.951,173.236,45.875,159.106
C04357=1034.409,385.691,362.909,173.245,45.878,159.108
C04358=1034.418,385.937,362.867,173.252,45.882,159.110
C04359=1034.427,386.183,362.825,173.260,45.885,159.111
C04360=1034.436,386.429,362.783,173.269,45.889,159.113
C04361=1034.445,386.676,362.741,173.277,45.892,159.115
C04362=1034.455,386.921,362.699,173.286,45.896,159.117
C04363=1034.463,387.169,362.656,173.295,45.899,159.119
C04364=1034.473,387.414,362.613,173.303,45.903,159.121
C04365=1034.482,387.660,362.571,173.311,45.906,159.123
C04366=1034.490,387.907,362.529,173.320,45.910,159.125
C04367=1034.499,388.153,362.486,173.328,45.914,159.126
C04368=1034.509,388.399,362.443,173.336,45.918,159.128
C04369=1034.518,388.645,362.400,173.345,45.922,159.130
C04370=1034.527,388.891,362.358,173.353,45.925,159.132
C04371=1034.536,389.137,362.316,173.362,45.929,159.134
C04372=1034.545,389.383,362.272,173.370,45.932,159.136
C04373=1034.554,389.629,362.230,173.379,45.937,159.138
C04374=1034.563,389.875,362.187,173.388,45.940,159.140
C04375=1034.573,390.122,362.144,173.396,45.944,159.142
C04376=1034.582,390.367,362.101,173.405,45.948,159.144
C04377=1034.590,390.613,362.058,173.414,45.952,159.146
C04378=1034.600,390.860,362.016,173.422,45.955,159.148
C04379=1034.609,391.106,361.973,173.431,45.959,159.150
C04380=1034.618,391.352,361.929,173.441,45.963,159.152
C04381=1034.627,391.598,361.886,173.449,45.967,159.154
C04382=1034.636,391.844,361.843,173.458,45.971,159.156
C04383=1034.646,392.090,361.800,173.467,45.975,159.158
C04384=1034.655,392.336,361.757,173.475,45.979,159.160
C04385=1034.664,392.564,361.717,173.484,45.982,159.162
C04386=1034.672,392.793,361.676,173.492,45.986,159.164
C04387=1034.681,393.020,361.636,173.500,45.990,159.165
C04388=1034.690,393.249,361.596,173.509,45.993,159.167
C04389=1034.698,393.477,361.555,173.516,45.997,159.169
C04390=1034.707,393.706,361.515,173.525,46.001,159.171
C04391=1034.715,393.934,361.475,173.533,46.004,159.173
C04392=1034.725,394.162,361.435,173.542,46.008,159.175
C04393=1034.734,394.408,361.392,173.551,46.012,159.177
C04394=1034.743,394.654,361.348,173.560,46.017,159.179
C04395=1034.753,394.900,361.304,173.568,46.020,159.181
C04396=1034.762,395.145,361.260,173.578,46.024,159.183
C04397=1034.771,395.391,361.216,173.587,46.029,159.185
C04398=1034.781,395.638,361.172,173.596,46.033,159.188
C04399=1034.790,395.883,361.130,173.605,46.037,159.190
C04400=1034.799,396.129,361.086,173.615,46.041,159.192
C04401=1034.809,396.376,361.041,173.624,46.046,159.194
C04402=1034.818,396.622,360.997,173.633,46.050,159.196
C04403=1034.828,396.867,360.954,173.643,46.054,159.198
C04404=1034.837,397.112,360.909,173.652,46.058,159.200
C04405=1034.847,397.358,360.865,173.661,46.062,159.203
C04406=1034.856,397.605,360.821,173.670,46.066,159.205
C04407=1034.866,397.850,360.778,173.680,46.071,159.207
C04408=1034.876,398.097,360.733,173.690,46.075,159.209
C04409=1034.885,398.341,360.689,173.699,46.079,159.211
C04410=1034.894,398.587,360.645,173.707,46.084,159.213
C04411=1034.904,398.833,360.601,173.718,46.088,159.216
C04412=1034.914,399.079,360.557,173.727,46.092,159.218
C04413=1034.924,399.325,360.512,173.736,46.096,159.220
C04414=1034.933,399.571,360.468,173.746,46.101,159.222
C04415=1034.943,399.817,360.424,173.756,46.105,159.225
C04416=1034.952,400.063,360.379,173.765,46.110,159.227
C04417=1034.963,400.308,360.335,173.775,46.115,159.229
C04418=1034.972,400.553,360.290,173.784,46.119,159.232
C04419=1034.982,400.800,360.246,173.794,46.123,159.234
C04420=1034.991,401.045,360.201,173.803,46.128,159.236
C04421=1035.002,401.291,360.156,173.813,46.132,159.238
C04422=1035.011,401.537,360.111,173.824,46.137,159.241
C04423=1035.021,401.783,360.067,173.833,46.141,159.243
C04424=1035.031,402.028,360.023,173.843,46.146,159.245
C04425=1035.040,402.274,359.978,173.852,46.151,159.248
C04426=1035.050,402.520,359.933,173.863,46.155,159.250
C04427=1035.060,402.766,359.888,173.873,46.160,159.253
C04428=1035.070,403.011,359.843,173.882,46.164,159.255
C04429=1035.079,403.257,359.797,173.892,46.169,159.257
C04430=1035.089,403.503,359.753,173.903,46.173,159.260
C04431=1035.099,403.749,359.707,173.912,46.178,159.262
C04432=1035.109,403.994,359.663,173.922,46.183,159.264
C04433=1035.119,404.239,359.617,173.933,46.188,159.267
C04434=1035.128,404.486,359.571,173.942,46.193,159.269
C04435=1035.138,404.731,359.526,173.952,46.197,159.272
C04436=1035.148,404.976,359.481,173.963,46.202,159.274
C04437=1035.158,405.222,359.436,173.973,46.207,159.277
C04438=1035.168,405.468,359.391,173.983,46.211,159.279
C04439=1035.178,405.714,359.344,173.993,46.216,159.282
C04440=1035.188,405.959,359.300,174.003,46.221,159.284
C04441=1035.198,406.205,359.254,174.013,46.226,159.287
C04442=1035.208,406.450,359.209,174.024,46.231,159.289
C04443=1035.219,406.696,359.163,174.034,46.236,159.291
C04444=1035.228,406.941,359.117,174.045,46.241,159.294
C04445=1035.238,407.180,359.073,174.054,46.245,159.296
C04446=1035.248,407.418,359.029,174.065,46.250,159.299
C04447=1035.258,407.657,358.984,174.075,46.255,159.301
C04448=1035.268,407.895,358.940,174.085,46.260,159.304
C04449=1035.277,408.134,358.895,174.095,46.265,159.306
C04450=1035.288,408.372,358.850,174.105,46.270,159.309
C04451=1035.298,408.611,358.806,174.116,46.274,159.311
C04452=1035.307,408.849,358.762,174.126,46.279,159.314
C04453=1035.318,409.095,358.716,174.137,46.284,159.316
C04454=1035.328,409.340,358.670,174.147,46.289,159.319
C04455=1035.338,409.586,358.624,174.158,46.294,159.322
C04456=1035.349,409.831,358.578,174.168,46.299,159.324
C04457=1035.359,410.077,358.532,174.179,46.305,159.327
C04458=1035.370,410.323,358.486,174.190,46.310,159.330
C04459=1035.380,410.568,358.439,174.201,46.314,159.332
C04460=1035.391,410.813,358.393,174.212,46.320,159.335
C04461=1035.401,411.059,358.347,174.223,46.325,159.338
C04462=1035.411,411.305,358.301,174.233,46.330,159.340
C04463=1035.422,411.550,358.254,174.244,46.335,159.343
C04464=1035.432,411.796,358.207,174.255,46.341,159.346
C04465=1035.443,412.041,358.161,174.267,46.346,159.348
C04466=1035.453,412.287,358.114,174.278,46.351,159.351
C04467=1035.464,412.532,358.068,174.289,46.357,159.354
C04468=1035.474,412.777,358.020,174.299,46.362,159.357
C04469=1035.485,413.023,357.975,174.311,46.367,159.359
C04470=1035.495,413.268,357.927,174.322,46.373,159.362
C04471=1035.505,413.513,357.880,174.333,46.378,159.365
C04472=1035.516,413.758,357.834,174.345,46.383,159.368
C04473=1035.526,414.004,357.787,174.356,46.389,159.371
C04474=1035.537,414.249,357.740,174.366,46.394,159.373
C04475=1035.547,414.495,357.693,174.378,46.400,159.376
C04476=1035.558,414.740,357.646,174.389,46.405,159.379
C04477=1035.569,414.985,357.599,174.401,46.410,159.382
C04478=1035.579,415.231,357.552,174.412,46.416,159.385
C04479=1035.590,415.476,357.505,174.424,46.422,159.388
C04480=1035.600,415.722,357.458,174.435,46.427,159.391
C04481=1035.612,415.966,357.410,174.447,46.433,159.394
C04482=1035.623,416.212,357.363,174.458,46.438,159.396
C04483=1035.633,416.457,357.316,174.470,46.444,159.399
C04484=1035.644,416.703,357.268,174.481,46.450,159.402
C04485=1035.655,416.947,357.221,174.493,46.455,159.405
C04486=1035.666,417.193,357.174,174.506,46.461,159.408
C04487=1035.676,417.438,357.126,174.517,46.467,159.411
C04488=1035.688,417.684,357.078,174.529,46.472,159.414
C04489=1035.698,417.929,357.031,174.541,46.477,159.417
C04490=1035.709,418.174,356.982,174.552,46.484,159.420
C04491=1035.720,418.419,356.935,174.564,46.489,159.423
C04492=1035.731,418.664,356.887,174.577,46.495,159.426
C04493=1035.741,418.909,356.840,174.588,46.501,159.429
C04494=1035.752,419.155,356.791,174.600,46.507,159.432
C04495=1035.763,419.399,356.743,174.612,46.512,159.435
C04496=1035.774,419.645,356.695,174.625,46.518,159.438
C04497=1035.786,419.890,356.647,174.637,46.524,159.442
C04498=1035.797,420.135,356.599,174.649,46.530,159.445
C04499=1035.808,420.380,356.551,174.661,46.536,159.448
C04500=1035.819,420.625,356.503,174.673,46.542,159.451
C04501=1035.830,420.871,356.455,174.685,46.548,159.454
C04502=1035.841,421.116,356.406,174.698,46.554,159.457
C04503=1035.851,421.361,356.358,174.710,46.560,159.460
C04504=1035.863,421.605,356.310,174.723,46.566,159.463
C04505=1035.875,421.863,356.259,174.735,46.573,159.467
C04506=1035.886,422.119,356.208,174.749,46.579,159.470
C04507=1035.899,422.376,356.158,174.762,46.585,159.473
C04508=1035.910,422.633,356.107,174.775,46.591,159.477
C04509=1035.921,422.878,356.058,174.788,46.597,159.480
C04510=1035.933,423.123,356.010,174.801,46.604,159.483
C04511=1035.944,423.368,355.962,174.813,46.610,159.487
C04512=1035.956,423.613,355.913,174.826,46.616,159.490
C04513=1035.967,423.850,355.865,174.838,46.622,159.493
C04514=1035.978,424.087,355.817,174.851,46.628,159.496
C04515=1035.989,424.324,355.770,174.863,46.634,159.499
C04516=1036.000,424.561,355.723,174.876,46.640,159.503
C04517=1036.011,424.798,355.675,174.888,46.647,159.506
C04518=1036.022,425.035,355.627,174.901,46.653,159.509
C04519=1036.033,425.272,355.580,174.913,46.658,159.512
C04520=1036.044,425.508,355.533,174.926,46.665,159.516
C04521=1036.055,425.754,355.483,174.940,46.671,159.519
C04522=1036.067,425.999,355.434,174.953,46.678,159.523
C04523=1036.078,426.243,355.385,174.965,46.684,159.526
C04524=1036.090,426.488,355.335,174.979,46.690,159.529
C04525=1036.102,426.733,355.286,174.992,46.697,159.533
C04526=1036.113,426.977,355.236,175.006,46.703,159.536
C04527=1036.125,427.223,355.187,175.019,46.710,159.540
C04528=1036.137,427.467,355.138,175.033,46.716,159.543
C04529=1036.148,427.712,355.087,175.046,46.723,159.547
C04530=1036.160,427.957,355.038,175.060,46.730,159.550
C04531=1036.172,428.202,354.988,175.073,46.736,159.554
C04532=1036.183,428.446,354.938,175.087,46.743,159.557
C04533=1036.195,428.691,354.888,175.101,46.749,159.561
C04534=1036.207,428.936,354.839,175.114,46.756,159.565
C04535=1036.218,429.181,354.788,175.128,46.763,159.568
C04536=1036.230,429.425,354.738,175.142,46.770,159.572
C04537=1036.242,429.670,354.688,175.156,46.776,159.575
C04538=1036.253,429.915,354.638,175.169,46.783,159.579
C04539=1036.266,430.159,354.588,175.183,46.790,159.583
C04540=1036.278,430.404,354.538,175.197,46.796,159.586
C04541=1036.290,430.649,354.486,175.212,46.803,159.590
C04542=1036.302,430.893,354.437,175.226,46.810,159.594
C04543=1036.314,431.138,354.387,175.240,46.817,159.598
C04544=1036.326,431.383,354.336,175.254,46.824,159.601
C04545=1036.338,431.627,354.285,175.268,46.831,159.605
C04546=1036.350,431.872,354.235,175.282,46.838,159.609
C04547=1036.362,432.116,354.184,175.296,46.845,159.613
C04548=1036.374,432.360,354.134,175.311,46.852,159.616
C04549=1036.387,432.605,354.083,175.326,46.859,159.620
C04550=1036.398,432.850,354.032,175.341,46.865,159.624
C04551=1036.411,433.094,353.981,175.355,46.872,159.628
C04552=1036.423,433.338,353.931,175.369,46.880,159.632
C04553=1036.435,433.583,353.879,175.384,46.887,159.635
C04554=1036.449,433.828,353.828,175.398,46.894,159.639
C04555=1036.461,434.072,353.778,175.414,46.901,159.643
C04556=1036.473,434.317,353.727,175.428,46.908,159.647
C04557=1036.485,434.561,353.676,175.443,46.915,159.651
C04558=1036.497,434.806,353.624,175.458,46.922,159.655
C04559=1036.511,435.050,353.572,175.473,46.929,159.659
C04560=1036.523,435.294,353.521,175.488,46.937,159.663
C04561=1036.535,435.539,353.470,175.503,46.944,159.667
C04562=1036.547,435.782,353.418,175.518,46.952,159.671
C04563=1036.560,436.028,353.366,175.533,46.959,159.675
C04564=1036.573,436.272,353.316,175.549,46.966,159.679
C04565=1036.585,436.516,353.263,175.564,46.974,159.683
C04566=1036.598,436.759,353.212,175.579,46.981,159.687
C04567=1036.611,437.003,353.160,175.595,46.988,159.692
C04568=1036.623,437.247,353.108,175.610,46.996,159.696
C04569=1036.636,437.490,353.057,175.626,47.003,159.700
C04570=1036.648,437.734,353.005,175.641,47.011,159.704
C04571=1036.661,437.979,352.953,175.657,47.018,159.708
C04572=1036.674,438.222,352.901,175.673,47.025,159.712
C04573=1036.687,438.466,352.849,175.689,47.033,159.717
C04574=1036.699,438.711,352.797,175.704,47.041,159.721
C04575=1036.712,438.955,352.744,175.720,47.049,159.725
C04576=1036.725,439.199,352.693,175.736,47.056,159.729
C04577=1036.738,439.443,352.640,175.752,47.064,159.734
C04578=1036.751,439.687,352.587,175.768,47.072,159.738
C04579=1036.764,439.932,352.535,175.784,47.079,159.742
C04580=1036.777,440.175,352.483,175.801,47.087,159.747
C04581=1036.790,440.419,352.430,175.817,47.094,159.751
C04582=1036.803,440.664,352.377,175.833,47.102,159.755
C04583=1036.816,440.908,352.324,175.849,47.110,159.760
C04584=1036.829,441.152,352.271,175.866,47.118,159.764
C04585=1036.842,441.396,352.219,175.882,47.126,159.769
C04586=1036.855,441.640,352.166,175.898,47.134,159.773
C04587=1036.868,441.884,352.112,175.916,47.142,159.778
C04588=1036.882,442.128,352.059,175.932,47.150,159.782
C04589=1036.895,442.372,352.007,175.948,47.158,159.787
C04590=1036.908,442.616,351.953,175.965,47.166,159.791
C04591=1036.922,442.860,351.900,175.982,47.174,159.796
C04592=1036.935,443.104,351.847,175.999,47.182,159.800
C04593=1036.949,443.347,351.794,176.017,47.190,159.805
C04594=1036.963,443.591,351.740,176.033,47.198,159.810
C04595=1036.976,443.835,351.687,176.051,47.206,159.814
C04596=1036.989,444.079,351.633,176.067,47.214,159.819
C04597=1037.003,444.322,351.580,176.085,47.222,159.824
C04598=1037.017,444.564,351.528,176.101,47.230,159.828
C04599=1037.032,444.808,351.476,176.119,47.238,159.833
C04600=1037.047,445.053,351.423,176.137,47.246,159.837
C04601=1037.064,445.295,351.372,176.154,47.254,159.842
C04602=1037.080,445.539,351.321,176.172,47.261,159.846
C04603=1037.097,445.783,351.271,176.190,47.269,159.851
C04604=1037.114,446.027,351.221,176.208,47.276,159.856
C04605=1037.132,446.271,351.171,176.225,47.284,159.860
C04606=1037.151,446.514,351.122,176.243,47.291,159.865
C04607=1037.170,446.758,351.073,176.262,47.298,159.869
C04608=1037.190,447.003,351.024,176.279,47.305,159.874
C04609=1037.210,447.247,350.977,176.297,47.312,159.878
C04610=1037.231,447.492,350.930,176.316,47.319,159.883
C04611=1037.253,447.736,350.883,176.334,47.325,159.887
C04612=1037.275,447.981,350.836,176.353,47.332,159.892
C04613=1037.297,448.225,350.790,176.371,47.339,159.896
C04614=1037.320,448.470,350.744,176.390,47.346,159.901
C04615=1037.344,448.715,350.699,176.409,47.352,159.905
C04616=1037.368,448.960,350.654,176.428,47.358,159.909
C04617=1037.392,449.205,350.610,176.446,47.365,159.914
C04618=1037.418,449.450,350.566,176.465,47.371,159.918
C04619=1037.443,449.695,350.523,176.484,47.377,159.923
C04620=1037.470,449.939,350.480,176.503,47.383,159.927
C04621=1037.497,450.185,350.437,176.523,47.389,159.931
C04622=1037.524,450.430,350.396,176.542,47.395,159.936
C04623=1037.552,450.676,350.353,176.561,47.401,159.940
C04624=1037.580,450.921,350.313,176.580,47.406,159.944
C04625=1037.620,451.251,350.258,176.606,47.414,159.950
C04626=1037.660,451.580,350.205,176.633,47.421,159.956
C04627=1037.700,451.908,350.152,176.660,47.428,159.962
C04628=1037.742,452.237,350.100,176.686,47.436,159.967
C04629=1037.451,452.292,349.777,176.689,47.507,159.990
C04630=1037.411,451.977,349.826,176.663,47.501,159.984
C04631=1037.372,451.661,349.877,176.638,47.494,159.979
C04632=1037.332,451.346,349.928,176.613,47.487,159.973
C04633=1037.295,451.030,349.980,176.588,47.479,159.968
C04634=1037.266,450.785,350.021,176.568,47.474,159.963
C04635=1037.237,450.539,350.062,176.548,47.469,159.959
C04636=1037.210,450.294,350.104,176.529,47.462,159.955
C04637=1037.183,450.048,350.147,176.510,47.457,159.950
C04638=1037.156,449.803,350.189,176.490,47.451,159.946
C04639=1037.130,449.558,350.232,176.471,47.445,159.942
C04640=1037.105,449.314,350.275,176.452,47.439,159.937
C04641=1037.079,449.069,350.320,176.433,47.433,159.933
C04642=1037.055,448.823,350.364,176.415,47.426,159.928
C04643=1037.031,448.579,350.409,176.396,47.420,159.924
C04644=1037.008,448.334,350.454,176.377,47.414,159.920
C04645=1036.985,448.089,350.501,176.359,47.407,159.915
C04646=1036.963,447.845,350.546,176.340,47.401,159.911
C04647=1036.941,447.601,350.593,176.321,47.394,159.906
C04648=1036.920,447.355,350.640,176.303,47.387,159.902
C04649=1036.899,447.111,350.688,176.285,47.380,159.897
C04650=1036.879,446.867,350.737,176.267,47.374,159.893
C04651=1036.860,446.622,350.785,176.248,47.367,159.888
C04652=1036.841,446.378,350.834,176.231,47.359,159.884
C04653=1036.822,446.135,350.883,176.212,47.352,159.879
C04654=1036.805,445.891,350.933,176.195,47.345,159.875
C04655=1036.787,445.646,350.983,176.176,47.338,159.870
C04656=1036.770,445.403,351.034,176.159,47.330,159.865
C04657=1036.754,445.160,351.085,176.142,47.323,159.861
C04658=1036.739,444.916,351.136,176.124,47.315,159.856
C04659=1036.723,444.672,351.189,176.106,47.307,159.852
C04660=1036.709,444.429,351.241,176.089,47.300,159.847
C04661=1036.694,444.187,351.294,176.072,47.291,159.842
C04662=1036.681,443.943,351.347,176.055,47.283,159.838
C04663=1036.666,443.699,351.401,176.037,47.276,159.833
C04664=1036.653,443.456,351.454,176.020,47.267,159.828
C04665=1036.640,443.212,351.507,176.003,47.260,159.824
C04666=1036.627,442.968,351.561,175.986,47.251,159.819
C04667=1036.613,442.725,351.614,175.970,47.243,159.815
C04668=1036.600,442.481,351.667,175.952,47.236,159.810
C04669=1036.586,442.236,351.720,175.936,47.227,159.806
C04670=1036.573,441.992,351.773,175.918,47.220,159.801
C04671=1036.559,441.748,351.826,175.902,47.212,159.797
C04672=1036.546,441.504,351.879,175.886,47.204,159.792
C04673=1036.533,441.260,351.932,175.869,47.196,159.788
C04674=1036.521,441.016,351.985,175.852,47.189,159.783
C04675=1036.508,440.772,352.038,175.836,47.181,159.779
C04676=1036.494,440.528,352.090,175.819,47.173,159.774
C04677=1036.481,440.284,352.143,175.803,47.166,159.770
C04678=1036.468,440.040,352.195,175.787,47.158,159.766
C04679=1036.455,439.796,352.249,175.771,47.150,159.761
C04680=1036.442,439.551,352.301,175.754,47.142,159.757
C04681=1036.430,439.307,352.353,175.738,47.135,159.753
C04682=1036.416,439.064,352.406,175.722,47.127,159.748
C04683=1036.403,438.819,352.458,175.706,47.120,159.744
C04684=1036.391,438.575,352.510,175.690,47.112,159.740
C04685=1036.378,438.331,352.562,175.675,47.105,159.736
C04686=1036.364,438.086,352.614,175.659,47.097,159.732
C04687=1036.352,437.843,352.666,175.643,47.090,159.727
C04688=1036.339,437.598,352.719,175.628,47.083,159.723
C04689=1036.327,437.354,352.770,175.613,47.075,159.719
C04690=1036.314,437.109,352.822,175.597,47.067,159.715
C04691=1036.301,436.865,352.875,175.581,47.060,159.711
C04692=1036.289,436.619,352.926,175.566,47.053,159.707
C04693=1036.276,436.374,352.978,175.550,47.046,159.703
C04694=1036.263,436.131,353.030,175.535,47.039,159.698
C04695=1036.251,435.886,353.081,175.519,47.031,159.694
C04696=1036.238,435.642,353.133,175.504,47.024,159.690
C04697=1036.226,435.397,353.184,175.489,47.017,159.686
C04698=1036.213,435.153,353.235,175.474,47.009,159.682
C04699=1036.201,434.909,353.287,175.459,47.002,159.678
C04700=1036.189,434.665,353.338,175.444,46.995,159.674
C04701=1036.176,434.420,353.390,175.429,46.988,159.670
C04702=1036.164,434.176,353.441,175.414,46.981,159.667
C04703=1036.151,433.931,353.492,175.399,46.974,159.663
C04704=1036.139,433.687,353.543,175.385,46.967,159.659
C04705=1036.127,433.442,353.593,175.370,46.960,159.655
C04706=1036.114,433.198,353.644,175.355,46.953,159.651
C04707=1036.102,432.953,353.695,175.341,46.946,159.647
C04708=1036.090,432.709,353.746,175.326,46.939,159.643
C04709=1036.077,432.464,353.796,175.312,46.932,159.639
C04710=1036.065,432.220,353.848,175.297,46.926,159.636
C04711=1036.053,431.975,353.898,175.282,46.919,159.632
C04712=1036.040,431.731,353.948,175.268,46.912,159.628
C04713=1036.029,431.486,353.999,175.254,46.905,159.624
C04714=1036.017,431.241,354.049,175.239,46.898,159.621
C04715=1036.004,430.997,354.100,175.225,46.891,159.617
C04716=1035.993,430.752,354.150,175.211,46.884,159.613
C04717=1035.981,430.507,354.200,175.197,46.877,159.609
C04718=1035.968,430.263,354.251,175.183,46.871,159.606
C04719=1035.957,430.018,354.302,175.169,46.864,159.602
C04720=1035.945,429.774,354.352,175.155,46.857,159.598
C04721=1035.932,429.529,354.402,175.141,46.851,159.595
C04722=1035.921,429.284,354.452,175.127,46.844,159.591
C04723=1035.909,429.040,354.502,175.114,46.837,159.588
C04724=1035.897,428.794,354.552,175.100,46.831,159.584
C04725=1035.886,428.550,354.602,175.086,46.825,159.580
C04726=1035.874,428.305,354.652,175.072,46.817,159.577
C04727=1035.862,428.061,354.702,175.058,46.811,159.573
C04728=1035.851,427.815,354.752,175.044,46.805,159.570
C04729=1035.839,427.571,354.801,175.032,46.798,159.566
C04730=1035.827,427.326,354.851,175.018,46.792,159.563
C04731=1035.815,427.082,354.901,175.005,46.785,159.559
C04732=1035.803,426.836,354.950,174.991,46.779,159.556
C04733=1035.793,426.591,355.000,174.978,46.772,159.552
C04734=1035.781,426.346,355.050,174.964,46.766,159.549
C04735=1035.769,426.102,355.099,174.951,46.760,159.545
C04736=1035.758,425.857,355.148,174.937,46.753,159.542
C04737=1035.746,425.612,355.197,174.925,46.747,159.539
C04738=1035.734,425.367,355.246,174.911,46.741,159.535
C04739=1035.723,425.122,355.295,174.898,46.735,159.532
C04740=1035.711,424.877,355.344,174.886,46.728,159.529
C04741=1035.700,424.632,355.393,174.872,46.722,159.525
C04742=1035.689,424.388,355.442,174.859,46.716,159.522
C04743=1035.677,424.143,355.491,174.847,46.710,159.518
C04744=1035.665,423.897,355.541,174.834,46.703,159.515
C04745=1035.655,423.652,355.590,174.820,46.697,159.512
C04746=1035.643,423.409,355.638,174.808,46.691,159.509
C04747=1035.632,423.165,355.687,174.795,46.685,159.505
C04748=1035.621,422.921,355.735,174.782,46.679,159.502
C04749=1035.609,422.677,355.783,174.770,46.673,159.499
C04750=1035.598,422.432,355.832,174.758,46.667,159.496
C04751=1035.586,422.189,355.880,174.745,46.661,159.492
C04752=1035.575,421.945,355.929,174.732,46.655,159.489
C04753=1035.564,421.700,355.976,174.719,46.649,159.486
C04754=1035.553,421.456,356.025,174.707,46.644,159.483
C04755=1035.542,421.210,356.073,174.694,46.637,159.480
C04756=1035.531,420.965,356.122,174.682,46.632,159.477
C04757=1035.520,420.720,356.170,174.670,46.626,159.473
C04758=1035.509,420.475,356.218,174.657,46.620,159.470
C04759=1035.497,420.230,356.266,174.646,46.614,159.467
C04760=1035.486,419.984,356.314,174.634,46.608,159.464
C04761=1035.476,419.740,356.362,174.621,46.602,159.461
C04762=1035.464,419.494,356.410,174.609,46.597,159.458
C04763=1035.453,419.249,356.458,174.597,46.591,159.455
C04764=1035.443,419.004,356.506,174.584,46.585,159.452
C04765=1035.432,418.759,356.555,174.572,46.579,159.449
C04766=1035.420,418.514,356.602,174.561,46.573,159.446
C04767=1035.410,418.269,356.649,174.549,46.568,159.443
C04768=1035.399,418.023,356.698,174.536,46.562,159.440
C04769=1035.388,417.779,356.746,174.524,46.556,159.437
C04770=1035.377,417.533,356.793,174.513,46.551,159.434
C04771=1035.367,417.288,356.841,174.501,46.545,159.431
C04772=1035.355,417.042,356.888,174.489,46.539,159.428
C04773=1035.345,416.797,356.935,174.478,46.534,159.425
C04774=1035.329,416.454,357.002,174.461,46.526,159.421
C04775=1035.314,416.111,357.069,174.444,46.518,159.417
C04776=1035.300,415.767,357.134,174.429,46.511,159.413
C04777=1035.284,415.424,357.200,174.412,46.503,159.408
C04778=1035.274,415.179,357.248,174.401,46.498,159.406
C04779=1035.262,414.933,357.295,174.389,46.492,159.403
C04780=1035.252,414.688,357.342,174.378,46.487,159.400
C04781=1035.241,414.443,357.389,174.366,46.482,159.397
C04782=1035.231,414.198,357.436,174.355,46.476,159.394
C04783=1035.220,413.951,357.483,174.343,46.471,159.391
C04784=1035.210,413.706,357.529,174.333,46.465,159.389
C04785=1035.199,413.461,357.577,174.322,46.460,159.386
C04786=1035.188,413.216,357.623,174.310,46.455,159.383
C04787=1035.178,412.971,357.670,174.299,46.449,159.380
C04788=1035.168,412.725,357.716,174.288,46.444,159.378
C04789=1035.157,412.480,357.763,174.276,46.439,159.375
C04790=1035.147,412.234,357.809,174.265,46.433,159.372
C04791=1035.137,411.989,357.857,174.255,46.428,159.369
C04792=1035.126,411.744,357.903,174.243,46.423,159.367
C04793=1035.116,411.498,357.950,174.232,46.418,159.364
C04794=1035.106,411.252,357.996,174.221,46.413,159.361
C04795=1035.095,411.007,358.043,174.211,46.408,159.358
C04796=1035.084,410.761,358.089,174.199,46.403,159.356
C04797=1035.074,410.516,358.135,174.188,46.397,159.353
C04798=1035.064,410.270,358.181,174.178,46.392,159.350
C04799=1035.053,410.025,358.228,174.167,46.387,159.348
C04800=1035.042,409.779,358.274,174.156,46.382,159.345
C04801=1035.032,409.534,358.320,174.146,46.377,159.343
C04802=1035.022,409.288,358.366,174.135,46.372,159.340
C04803=1035.012,409.043,358.412,174.124,46.368,159.337
C04804=1035.001,408.797,358.458,174.113,46.363,159.335
C04805=1034.990,408.552,358.503,174.102,46.358,159.332
C04806=1034.975,408.170,358.574,174.086,46.350,159.328
C04807=1034.959,407.790,358.645,174.069,46.342,159.324
C04808=1034.943,407.409,358.717,174.054,46.335,159.320
C04809=1034.928,407.028,358.787,174.038,46.327,159.316
C04810=1034.918,406.782,358.833,174.027,46.322,159.314
C04811=1034.907,406.536,358.878,174.017,46.318,159.311
C04812=1034.897,406.291,358.924,174.006,46.313,159.309
C04813=1034.887,406.045,358.969,173.996,46.308,159.306
C04814=1034.878,405.800,359.015,173.985,46.303,159.304
C04815=1034.867,405.554,359.060,173.975,46.299,159.301
C04816=1034.857,405.309,359.106,173.966,46.294,159.299
C04817=1034.848,405.063,359.151,173.955,46.289,159.296
C04818=1034.837,404.818,359.197,173.945,46.285,159.294
C04819=1034.827,404.572,359.242,173.935,46.280,159.292
C04820=1034.818,404.326,359.287,173.924,46.275,159.289
C04821=1034.808,404.080,359.332,173.915,46.270,159.287
C04822=1034.798,403.835,359.378,173.905,46.266,159.284
C04823=1034.788,403.589,359.423,173.894,46.261,159.282
C04824=1034.778,403.343,359.468,173.884,46.257,159.280
C04825=1034.769,403.098,359.513,173.875,46.252,159.277
C04826=1034.759,402.852,359.558,173.865,46.247,159.275
C04827=1034.749,402.606,359.603,173.854,46.243,159.272
C04828=1034.739,402.360,359.648,173.845,46.238,159.270
C04829=1034.729,402.115,359.693,173.835,46.234,159.268
C04830=1034.720,401.869,359.738,173.825,46.229,159.265
C04831=1034.710,401.624,359.782,173.816,46.225,159.263
C04832=1034.700,401.377,359.827,173.805,46.220,159.261
C04833=1034.690,401.131,359.872,173.795,46.216,159.258
C04834=1034.681,400.886,359.917,173.786,46.211,159.256
C04835=1034.671,400.640,359.961,173.776,46.207,159.254
C04836=1034.662,400.394,360.005,173.767,46.202,159.252
C04837=1034.652,400.149,360.050,173.757,46.198,159.249
C04838=1034.642,399.903,360.094,173.747,46.194,159.247
C04839=1034.632,399.657,360.139,173.738,46.190,159.245
C04840=1034.623,399.411,360.183,173.728,46.185,159.242
C04841=1034.613,399.166,360.228,173.718,46.181,159.240
C04842=1034.603,398.920,360.272,173.709,46.177,159.238
C04843=1034.594,398.674,360.317,173.699,46.172,159.236
C04844=1034.584,398.428,360.360,173.690,46.168,159.234
C04845=1034.574,398.182,360.404,173.680,46.164,159.231
C04846=1034.564,397.937,360.449,173.671,46.160,159.229
C04847=1034.555,397.691,360.493,173.661,46.156,159.227
C04848=1034.545,397.445,360.536,173.652,46.151,159.225
C04849=1034.536,397.199,360.580,173.643,46.148,159.223
C04850=1034.527,396.953,360.624,173.634,46.143,159.221
C04851=1034.517,396.707,360.669,173.625,46.139,159.218
C04852=1034.507,396.461,360.712,173.615,46.135,159.216
C04853=1034.498,396.216,360.756,173.606,46.131,159.214
C04854=1034.489,395.970,360.800,173.597,46.127,159.212
C04855=1034.479,395.724,360.843,173.587,46.123,159.210
C04856=1034.469,395.478,360.888,173.578,46.118,159.208
C04857=1034.460,395.232,360.931,173.569,46.114,159.205
C04858=1034.451,394.986,360.975,173.559,46.110,159.203
C04859=1034.441,394.740,361.019,173.550,46.106,159.201
C04860=1034.432,394.495,361.063,173.542,46.102,159.199
C04861=1034.423,394.248,361.106,173.533,46.098,159.197
C04862=1034.414,394.019,361.147,173.524,46.094,159.195
C04863=1034.405,393.790,361.187,173.516,46.091,159.193
C04864=1034.397,393.560,361.227,173.507,46.087,159.191
C04865=1034.388,393.331,361.268,173.498,46.084,159.189
C04866=1034.379,393.101,361.309,173.490,46.080,159.188
C04867=1034.370,392.872,361.349,173.482,46.076,159.186
C04868=1034.362,392.643,361.389,173.474,46.072,159.184
C04869=1034.353,392.414,361.430,173.465,46.069,159.182
C04870=1034.343,392.167,361.472,173.456,46.065,159.180
C04871=1034.335,391.922,361.516,173.448,46.061,159.178
C04872=1034.325,391.676,361.559,173.439,46.057,159.176
C04873=1034.316,391.430,361.602,173.430,46.053,159.174
C04874=1034.306,391.183,361.645,173.420,46.050,159.172
C04875=1034.298,390.938,361.689,173.412,46.046,159.170
C04876=1034.289,390.692,361.732,173.403,46.042,159.168
C04877=1034.279,390.445,361.774,173.395,46.038,159.166
C04878=1034.270,390.199,361.817,173.386,46.035,159.164
C04879=1034.261,389.953,361.860,173.377,46.031,159.162
C04880=1034.252,389.707,361.903,173.369,46.027,159.160
C04881=1034.243,389.461,361.946,173.360,46.024,159.158
C04882=1034.234,389.215,361.988,173.352,46.020,159.156
C04883=1034.224,388.969,362.031,173.343,46.016,159.154
C04884=1034.216,388.723,362.074,173.334,46.012,159.152
C04885=1034.206,388.477,362.116,173.326,46.009,159.150
C04886=1034.197,388.230,362.160,173.317,46.005,159.148
C04887=1034.188,387.984,362.202,173.309,46.002,159.147
C04888=1034.179,387.739,362.245,173.300,45.998,159.145
C04889=1034.171,387.492,362.287,173.292,45.994,159.143
C04890=1034.161,387.246,362.329,173.283,45.990,159.141
C04891=1034.151,387.000,362.372,173.275,45.987,159.139
C04892=1034.143,386.753,362.414,173.266,45.984,159.137
C04893=1034.133,386.508,362.456,173.258,45.980,159.135
C04894=1034.124,386.261,362.498,173.249,45.977,159.134
C04895=1034.116,386.015,362.541,173.242,45.973,159.132
C04896=1034.106,385.768,362.583,173.233,45.969,159.130
C04897=1034.097,385.522,362.626,173.225,45.966,159.128
C04898=1034.088,385.276,362.667,173.216,45.963,159.126
C04899=1034.079,385.030,362.709,173.208,45.959,159.124
C04900=1034.070,384.784,362.751,173.200,45.956,159.123
C04901=1034.061,384.538,362.793,173.191,45.952,159.121
C04902=1034.052,384.291,362.835,173.184,45.949,159.119
C04903=1034.043,384.045,362.877,173.175,45.946,159.117
C04904=1034.035,383.799,362.920,173.167,45.943,159.116
C04905=1034.026,383.552,362.961,173.158,45.939,159.114
C04906=1034.017,383.306,363.003,173.150,45.936,159.112
C04907=1034.008,383.060,363.045,173.143,45.932,159.110
C04908=1033.999,382.813,363.086,173.135,45.929,159.108
C04909=1033.990,382.567,363.128,173.126,45.926,159.107
C04910=1033.981,382.321,363.171,173.118,45.923,159.105
C04911=1033.972,382.076,363.212,173.111,45.919,159.103
C04912=1033.963,381.829,363.254,173.102,45.916,159.102
C04913=1033.955,381.582,363.295,173.094,45.913,159.100
C04914=1033.946,381.336,363.336,173.087,45.909,159.098
C04915=1033.938,381.089,363.379,173.078,45.906,159.096
C04916=1033.929,380.843,363.420,173.070,45.903,159.095
C04917=1033.920,380.597,363.462,173.062,45.900,159.093
C04918=1033.912,380.351,363.503,173.054,45.896,159.091
C04919=1033.903,380.104,363.545,173.046,45.894,159.090
C04920=1033.894,379.857,363.586,173.039,45.890,159.088
C04921=1033.886,379.612,363.628,173.031,45.887,159.086
C04922=1033.878,379.399,363.664,173.024,45.884,159.085
C04923=1033.870,379.188,363.699,173.017,45.882,159.083
C04924=1033.863,378.976,363.735,173.011,45.879,159.082
C04925=1033.857,378.764,363.770,173.004,45.876,159.080
C04926=1033.848,378.552,363.806,172.997,45.873,159.079
C04927=1033.841,378.340,363.842,172.990,45.871,159.077
C04928=1033.834,378.129,363.877,172.984,45.868,159.076
C04929=1033.827,377.917,363.912,172.978,45.865,159.075
C04930=1033.818,377.670,363.954,172.970,45.862,159.073
C04931=1033.809,377.424,363.994,172.961,45.859,159.071
C04932=1033.801,377.177,364.035,172.954,45.856,159.070
C04933=1033.792,376.931,364.077,172.946,45.853,159.068
C04934=1033.783,376.684,364.118,172.939,45.850,159.067
C04935=1033.774,376.438,364.158,172.931,45.848,159.065
C04936=1033.766,376.191,364.199,172.924,45.844,159.063
C04937=1033.757,375.945,364.240,172.916,45.841,159.062
C04938=1033.749,375.698,364.281,172.909,45.839,159.060
C04939=1033.740,375.452,364.321,172.901,45.836,159.059
C04940=1033.731,375.205,364.362,172.893,45.832,159.057
C04941=1033.723,374.959,364.403,172.885,45.830,159.056
C04942=1033.715,374.712,364.444,172.878,45.827,159.054
C04943=1033.706,374.466,364.484,172.870,45.824,159.052
C04944=1033.697,374.219,364.525,172.863,45.821,159.051
C04945=1033.689,373.973,364.565,172.856,45.818,159.049
C04946=1033.680,373.726,364.606,172.848,45.816,159.048
C04947=1033.672,373.480,364.646,172.841,45.812,159.046
C04948=1033.664,373.234,364.687,172.833,45.810,159.045
C04949=1033.655,372.987,364.728,172.826,45.807,159.043
C04950=1033.646,372.741,364.768,172.819,45.804,159.042
C04951=1033.638,372.495,364.809,172.811,45.801,159.040
C04952=1033.630,372.247,364.849,172.804,45.799,159.039
C04953=1033.621,372.001,364.889,172.796,45.796,159.037
C04954=1033.613,371.755,364.930,172.789,45.793,159.036
C04955=1033.605,371.508,364.971,172.782,45.790,159.034
C04956=1033.597,371.261,365.010,172.774,45.788,159.033
C04957=1033.588,371.015,365.051,172.767,45.785,159.031
C04958=1033.580,370.768,365.091,172.760,45.782,159.030
C04959=1033.572,370.521,365.131,172.754,45.779,159.028
C04960=1033.563,370.275,365.171,172.746,45.777,159.027
C04961=1033.555,370.028,365.211,172.739,45.774,159.025
C04962=1033.547,369.782,365.252,172.732,45.771,159.024
C04963=1033.539,369.535,365.291,172.724,45.769,159.022
C04964=1033.530,369.288,365.332,172.717,45.766,159.021
C04965=1033.522,369.042,365.372,172.710,45.764,159.020
C04966=1033.514,368.795,365.412,172.703,45.761,159.018
C04967=1033.505,368.549,365.452,172.696,45.758,159.017
C04968=1033.497,368.302,365.491,172.689,45.756,159.015
C04969=1033.489,368.055,365.531,172.682,45.753,159.014
C04970=1033.480,367.808,365.571,172.675,45.750,159.012
C04971=1033.471,367.562,365.611,172.667,45.748,159.011
C04972=1033.463,367.315,365.651,172.660,45.745,159.010
C04973=1033.455,367.068,365.690,172.654,45.743,159.008
C04974=1033.447,366.821,365.730,172.647,45.741,159.007
C04975=1033.439,366.575,365.769,172.640,45.738,159.005
C04976=1033.430,366.328,365.808,172.632,45.735,159.004
C04977=1033.423,366.081,365.848,172.625,45.733,159.003
C04978=1033.414,365.835,365.888,172.619,45.731,159.001
C04979=1033.406,365.588,365.927,172.612,45.728,159.000
C04980=1033.398,365.341,365.967,172.605,45.725,158.999
C04981=1033.390,365.095,366.006,172.598,45.723,158.997
C04982=1033.376,364.692,366.072,172.586,45.719,158.995
C04983=1033.363,364.289,366.136,172.576,45.715,158.993
C04984=1033.350,363.886,366.199,172.565,45.711,158.991
C04985=1033.336,363.482,366.264,172.553,45.708,158.988
C04986=1033.328,363.236,366.303,172.546,45.705,158.987
C04987=1033.321,362.990,366.343,172.540,45.703,158.986
C04988=1033.313,362.742,366.381,172.533,45.700,158.985
C04989=1033.305,362.495,366.421,172.526,45.698,158.983
C04990=1033.296,362.249,366.461,172.519,45.696,158.982
C04991=1033.288,362.002,366.499,172.513,45.693,158.981
C04992=1033.281,361.755,366.539,172.506,45.691,158.979
C04993=1033.273,361.509,366.578,172.499,45.689,158.978
C04994=1033.265,361.262,366.617,172.493,45.686,158.977
C04995=1033.256,361.015,366.656,172.486,45.684,158.975
C04996=1033.249,360.768,366.694,172.480,45.682,158.974
C04997=1033.240,360.521,366.733,172.473,45.680,158.973
C04998=1033.233,360.274,366.773,172.466,45.677,158.972
C04999=1033.225,360.027,366.811,172.459,45.675,158.970
C05000=1033.217,359.781,366.850,172.453,45.673,158.969
C05001=1033.209,359.534,366.889,172.446,45.671,158.968
C05002=1033.200,359.287,366.928,172.440,45.668,158.967
C05003=1033.192,359.040,366.966,172.433,45.667,158.965
C05004=1033.184,358.794,367.005,172.427,45.664,158.964
C05005=1033.176,358.547,367.044,172.420,45.663,158.963
C05006=1033.168,358.299,367.082,172.413,45.660,158.962
C05007=1033.160,358.053,367.121,172.407,45.658,158.961
C05008=1033.152,357.806,367.159,172.400,45.656,158.959
C05009=1033.144,357.558,367.198,172.394,45.654,158.958
C05010=1033.137,357.312,367.236,172.387,45.652,158.957
C05011=1033.128,357.065,367.275,172.381,45.650,158.956
C05012=1033.121,356.819,367.314,172.374,45.648,158.954
C05013=1033.112,356.572,367.352,172.368,45.646,158.953
C05014=1033.105,356.325,367.391,172.362,45.643,158.952
C05015=1033.097,356.078,367.429,172.356,45.641,158.951
C05016=1033.089,355.831,367.468,172.349,45.640,158.950
C05017=1033.081,355.583,367.505,172.342,45.637,158.948
C05018=1033.073,355.336,367.544,172.336,45.635,158.947
C05019=1033.066,355.090,367.582,172.330,45.634,158.946
C05020=1033.058,354.842,367.621,172.323,45.631,158.945
C05021=1033.049,354.596,367.658,172.317,45.629,158.944
C05022=1033.041,354.348,367.696,172.311,45.627,158.943
C05023=1033.034,354.102,367.735,172.305,45.626,158.941
C05024=1033.026,353.855,367.773,172.298,45.624,158.940
C05025=1033.018,353.608,367.811,172.292,45.622,158.939
C05026=1033.011,353.361,367.849,172.285,45.620,158.938
C05027=1033.002,353.114,367.887,172.279,45.618,158.937
C05028=1032.995,352.867,367.924,172.273,45.616,158.936
C05029=1032.987,352.620,367.963,172.267,45.614,158.935
C05030=1032.979,352.373,368.001,172.261,45.612,158.933
C05031=1032.972,352.126,368.039,172.254,45.610,158.932
C05032=1032.963,351.879,368.077,172.248,45.609,158.931
C05033=1032.956,351.632,368.114,172.242,45.606,158.930
C05034=1032.948,351.385,368.153,172.236,45.605,158.929
C05035=1032.940,351.138,368.190,172.230,45.603,158.928
C05036=1032.933,350.891,368.229,172.223,45.601,158.927
C05037=1032.925,350.644,368.266,172.218,45.599,158.926
C05038=1032.912,350.247,368.327,172.207,45.596,158.924
C05039=1032.900,349.850,368.387,172.197,45.593,158.922
C05040=1032.888,349.453,368.448,172.188,45.591,158.920
C05041=1032.875,349.057,368.509,172.178,45.588,158.919
C05042=1032.868,348.810,368.546,172.173,45.586,158.917
C05043=1032.860,348.563,368.583,172.166,45.584,158.916
C05044=1032.852,348.316,368.621,172.160,45.583,158.915
C05045=1032.845,348.068,368.659,172.155,45.581,158.914
C05046=1032.837,347.821,368.696,172.148,45.579,158.913
C05047=1032.829,347.574,368.733,172.142,45.578,158.912
C05048=1032.821,347.327,368.770,172.136,45.576,158.911
C05049=1032.814,347.080,368.808,172.130,45.574,158.910
C05050=1032.806,346.833,368.844,172.124,45.572,158.909
C05051=1032.798,346.585,368.882,172.118,45.571,158.908
C05052=1032.790,346.338,368.919,172.113,45.569,158.907
C05053=1032.783,346.091,368.957,172.106,45.567,158.906
C05054=1032.775,345.844,368.994,172.101,45.566,158.905
C05055=1032.768,345.597,369.031,172.095,45.564,158.904
C05056=1032.760,345.351,369.068,172.089,45.563,158.903
C05057=1032.753,345.103,369.106,172.083,45.561,158.902
C05058=1032.745,344.856,369.143,172.077,45.560,158.901
C05059=1032.737,344.609,369.180,172.071,45.558,158.900
C05060=1032.730,344.362,369.217,172.066,45.556,158.899
C05061=1032.722,344.115,369.254,172.059,45.554,158.898
C05062=1032.714,343.868,369.291,172.054,45.553,158.897
C05063=1032.708,343.620,369.328,172.048,45.552,158.896
C05064=1032.700,343.373,369.365,172.041,45.550,158.895
C05065=1032.692,343.126,369.402,172.036,45.548,158.894
C05066=1032.685,342.879,369.438,172.030,45.547,158.893
C05067=1032.677,342.632,369.476,172.025,45.545,158.892
C05068=1032.669,342.385,369.513,172.019,45.544,158.891
C05069=1032.662,342.137,369.550,172.014,45.542,158.890
C05070=1032.655,341.890,369.587,172.007,45.541,158.889
C05071=1032.647,341.643,369.623,172.002,45.539,158.888
C05072=1032.640,341.396,369.660,171.996,45.538,158.887
C05073=1032.632,341.148,369.697,171.990,45.537,158.886
C05074=1032.625,340.901,369.734,171.985,45.535,158.885
C05075=1032.617,340.654,369.770,171.978,45.533,158.884
C05076=1032.609,340.407,369.807,171.973,45.532,158.883
C05077=1032.601,340.159,369.843,171.967,45.531,158.882
C05078=1032.594,339.913,369.879,171.962,45.529,158.881
C05079=1032.587,339.666,369.917,171.956,45.528,158.880
C05080=1032.579,339.418,369.953,171.951,45.526,158.879
C05081=1032.572,339.171,369.989,171.945,45.525,158.879
C05082=1032.564,338.923,370.025,171.939,45.524,158.878
C05083=1032.556,338.676,370.062,171.933,45.523,158.877
C05084=1032.550,338.429,370.099,171.928,45.521,158.876
C05085=1032.542,338.182,370.135,171.922,45.520,158.875
C05086=1032.534,337.934,370.171,171.917,45.518,158.874
C05087=1032.527,337.687,370.207,171.911,45.517,158.873
C05088=1032.519,337.440,370.244,171.906,45.516,158.872
C05089=1032.512,337.193,370.280,171.900,45.514,158.871
C05090=1032.505,336.946,370.317,171.895,45.514,158.870
C05091=1032.497,336.698,370.353,171.890,45.512,158.870
C05092=1032.489,336.451,370.389,171.883,45.511,158.869
C05093=1032.482,336.204,370.425,171.878,45.509,158.868
C05094=1032.470,335.803,370.484,171.869,45.508,158.866
C05095=1032.458,335.404,370.543,171.860,45.506,158.865
C05096=1032.447,335.004,370.601,171.851,45.503,158.863
C05097=1032.434,334.603,370.659,171.842,45.501,158.862
C05098=1032.428,334.356,370.696,171.837,45.500,158.861
C05099=1032.420,334.109,370.731,171.831,45.499,158.860
C05100=1032.412,333.861,370.767,171.826,45.497,158.859
C05101=1032.405,333.614,370.803,171.821,45.496,158.859
C05102=1032.397,333.367,370.839,171.815,45.495,158.858
C05103=1032.390,333.120,370.874,171.810,45.494,158.857
C05104=1032.383,332.872,370.910,171.804,45.493,158.856
C05105=1032.375,332.625,370.947,171.799,45.492,158.855
C05106=1032.368,332.377,370.982,171.794,45.491,158.854
C05107=1032.361,332.130,371.018,171.788,45.489,158.853
C05108=1032.353,331.883,371.054,171.783,45.489,158.853
C05109=1032.346,331.635,371.089,171.777,45.487,158.852
C05110=1032.339,331.388,371.125,171.772,45.486,158.851
C05111=1032.331,331.141,371.161,171.767,45.485,158.850
C05112=1032.324,330.894,371.196,171.761,45.484,158.849
C05113=1032.316,330.646,371.232,171.756,45.483,158.848
C05114=1032.309,330.399,371.267,171.751,45.482,158.848
C05115=1032.302,330.152,371.304,171.745,45.481,158.847
C05116=1032.295,329.904,371.339,171.740,45.480,158.846
C05117=1032.287,329.657,371.375,171.735,45.478,158.845
C05118=1032.281,329.409,371.410,171.731,45.477,158.844
C05119=1032.273,329.161,371.446,171.725,45.477,158.844
C05120=1032.265,328.915,371.481,171.720,45.475,158.843
C05121=1032.258,328.667,371.516,171.715,45.474,158.842
C05122=1032.251,328.420,371.552,171.709,45.474,158.841
C05123=1032.244,328.173,371.587,171.704,45.472,158.840
C05124=1032.237,327.925,371.623,171.699,45.471,158.840
C05125=1032.229,327.678,371.657,171.693,45.471,158.839
C05126=1032.222,327.430,371.694,171.688,45.470,158.838
C05127=1032.214,327.183,371.728,171.683,45.469,158.837
C05128=1032.207,326.935,371.764,171.678,45.467,158.836
C05129=1032.199,326.688,371.798,171.672,45.467,158.836
C05130=1032.192,326.441,371.833,171.668,45.466,158.835
C05131=1032.184,326.193,371.868,171.663,45.465,158.834
C05132=1032.178,325.946,371.903,171.657,45.464,158.834
C05133=1032.169,325.698,371.938,171.652,45.463,158.833
C05134=1032.163,325.450,371.973,171.647,45.463,158.832
C05135=1032.155,325.203,372.008,171.642,45.462,158.831
C05136=1032.147,324.956,372.043,171.636,45.461,158.831
C05137=1032.140,324.708,372.078,171.632,45.460,158.830
C05138=1032.133,324.461,372.112,171.627,45.459,158.829
C05139=1032.125,324.213,372.148,171.622,45.458,158.828
C05140=1032.118,323.966,372.183,171.616,45.458,158.828
C05141=1032.111,323.719,372.218,171.611,45.457,158.827
C05142=1032.104,323.472,372.252,171.606,45.456,158.826
C05143=1032.097,323.223,372.287,171.602,45.455,158.825
C05144=1032.089,322.976,372.322,171.596,45.454,158.825
C05145=1032.082,322.729,372.356,171.591,45.453,158.824
C05146=1032.075,322.482,372.391,171.586,45.453,158.823
C05147=1032.067,322.234,372.426,171.581,45.452,158.823
C05148=1032.060,321.986,372.461,171.576,45.451,158.822
C05149=1032.053,321.739,372.495,171.571,45.450,158.821
C05150=1032.041,321.334,372.552,171.562,45.449,158.820
C05151=1032.029,320.929,372.609,171.555,45.448,158.819
C05152=1032.018,320.525,372.665,171.547,45.446,158.818
C05153=1032.006,320.120,372.722,171.538,45.445,158.817
C05154=1031.999,319.873,372.757,171.534,45.445,158.816
C05155=1031.992,319.625,372.791,171.529,45.444,158.815
C05156=1031.985,319.378,372.826,171.524,45.443,158.815
C05157=1031.977,319.130,372.861,171.518,45.443,158.814
C05158=1031.970,318.883,372.894,171.513,45.442,158.813
C05159=1031.963,318.635,372.930,171.509,45.441,158.812
C05160=1031.956,318.388,372.963,171.504,45.441,158.812
C05161=1031.949,318.140,372.998,171.499,45.440,158.811
C05162=1031.942,317.893,373.032,171.494,45.439,158.810
C05163=1031.934,317.645,373.067,171.490,45.438,158.810
C05164=1031.928,317.397,373.101,171.485,45.438,158.809
C05165=1031.920,317.150,373.136,171.480,45.437,158.808
C05166=1031.914,316.902,373.170,171.474,45.436,158.808
C05167=1031.906,316.655,373.205,171.470,45.436,158.807
C05168=1031.899,316.408,373.239,171.465,45.435,158.806
C05169=1031.893,316.160,373.273,171.460,45.435,158.806
C05170=1031.885,315.913,373.308,171.455,45.434,158.805
C05171=1031.879,315.665,373.342,171.451,45.433,158.804
C05172=1031.872,315.418,373.375,171.446,45.432,158.804
C05173=1031.865,315.171,373.410,171.441,45.432,158.803
C05174=1031.858,314.923,373.444,171.437,45.431,158.802
C05175=1031.851,314.675,373.478,171.432,45.430,158.802
C05176=1031.844,314.428,373.513,171.427,45.429,158.801
C05177=1031.837,314.180,373.547,171.422,45.429,158.800
C05178=1031.830,313.932,373.581,171.418,45.428,158.800
C05179=1031.823,313.684,373.615,171.413,45.428,158.799
C05180=1031.816,313.438,373.650,171.408,45.427,158.798
C05181=1031.809,313.190,373.683,171.404,45.427,158.798
C05182=1031.803,312.942,373.718,171.399,45.426,158.797
C05183=1031.796,312.695,373.752,171.394,45.425,158.797
C05184=1031.788,312.447,373.785,171.389,45.425,158.796
C05185=1031.782,312.200,373.820,171.385,45.424,158.795
C05186=1031.775,311.953,373.854,171.380,45.423,158.795
C05187=1031.769,311.705,373.888,171.375,45.423,158.794
C05188=1031.761,311.457,373.922,171.370,45.422,158.793
C05189=1031.755,311.210,373.956,171.366,45.422,158.793
C05190=1031.748,310.962,373.990,171.361,45.422,158.792
C05191=1031.741,310.714,374.023,171.357,45.421,158.792
C05192=1031.733,310.467,374.056,171.351,45.421,158.791
C05193=1031.725,310.219,374.090,171.346,45.420,158.790
C05194=1031.718,309.971,374.124,171.342,45.420,158.790
C05195=1031.712,309.724,374.157,171.337,45.420,158.789
C05196=1031.704,309.476,374.190,171.333,45.419,158.789
C05197=1031.697,309.229,374.223,171.328,45.419,158.788
C05198=1031.690,308.981,374.257,171.323,45.419,158.788
C05199=1031.683,308.734,374.291,171.319,45.419,158.787
C05200=1031.676,308.486,374.324,171.314,45.418,158.787
C05201=1031.668,308.238,374.357,171.309,45.417,158.786
C05202=1031.661,307.991,374.391,171.305,45.417,158.785
C05203=1031.655,307.743,374.424,171.300,45.417,158.785
C05204=1031.648,307.495,374.457,171.296,45.416,158.784
C05205=1031.640,307.248,374.491,171.291,45.416,158.784
C05206=1031.628,306.848,374.544,171.284,45.416,158.783
C05207=1031.617,306.448,374.598,171.276,45.415,158.782
C05208=1031.605,306.049,374.651,171.269,45.414,158.781
C05209=1031.594,305.649,374.705,171.262,45.414,158.780
C05210=1031.588,305.401,374.738,171.258,45.414,158.780
C05211=1031.581,305.154,374.772,171.253,45.413,158.779
C05212=1031.573,304.906,374.804,171.249,45.413,158.778
C05213=1031.567,304.659,374.838,171.244,45.413,158.778
C05214=1031.560,304.410,374.871,171.240,45.412,158.777
C05215=1031.552,304.163,374.905,171.235,45.412,158.777
C05216=1031.545,303.915,374.937,171.230,45.412,158.776
C05217=1031.538,303.668,374.971,171.226,45.412,158.776
C05218=1031.532,303.420,375.003,171.222,45.412,158.775
C05219=1031.525,303.172,375.036,171.217,45.412,158.775
C05220=1031.518,302.925,375.069,171.212,45.411,158.774
C05221=1031.511,302.677,375.102,171.208,45.411,158.774
C05222=1031.504,302.429,375.135,171.203,45.411,158.773
C05223=1031.497,302.182,375.168,171.200,45.410,158.773
C05224=1031.490,301.934,375.201,171.195,45.410,158.772
C05225=1031.483,301.686,375.234,171.191,45.410,158.772
C05226=1031.477,301.439,375.267,171.186,45.410,158.771
C05227=1031.469,301.191,375.300,171.182,45.410,158.771
C05228=1031.463,300.944,375.333,171.177,45.409,158.770
C05229=1031.456,300.695,375.366,171.173,45.409,158.769
C05230=1031.449,300.448,375.398,171.168,45.409,158.769
C05231=1031.442,300.200,375.432,171.165,45.409,158.769
C05232=1031.435,299.953,375.465,171.160,45.408,158.768
C05233=1031.429,299.704,375.498,171.156,45.408,158.767
C05234=1031.421,299.457,375.530,171.151,45.408,158.767
C05235=1031.415,299.210,375.563,171.147,45.408,158.767
C05236=1031.408,298.961,375.596,171.142,45.408,158.766
C05237=1031.401,298.714,375.628,171.138,45.407,158.765
C05238=1031.394,298.466,375.661,171.134,45.407,158.765
C05239=1031.388,298.219,375.695,171.130,45.407,158.765
C05240=1031.381,297.971,375.727,171.125,45.407,158.764
C05241=1031.374,297.723,375.760,171.121,45.407,158.763
C05242=1031.368,297.476,375.793,171.116,45.406,158.763
C05243=1031.361,297.228,375.825,171.113,45.406,158.763
C05244=1031.354,296.980,375.858,171.108,45.406,158.762
C05245=1031.347,296.732,375.891,171.103,45.406,158.761
C05246=1031.341,296.485,375.923,171.099,45.406,158.761
C05247=1031.333,296.237,375.956,171.095,45.406,158.761
C05248=1031.327,295.989,375.989,171.091,45.405,158.760
C05249=1031.321,295.741,376.021,171.087,45.406,158.760
C05250=1031.315,295.493,376.053,171.082,45.405,158.759
C05251=1031.307,295.245,376.086,171.078,45.406,158.759
C05252=1031.301,294.998,376.119,171.073,45.405,158.758
C05253=1031.295,294.750,376.151,171.070,45.405,158.758
C05254=1031.287,294.502,376.184,171.065,45.405,158.757
C05255=1031.281,294.255,376.217,171.061,45.405,158.757
C05256=1031.274,294.007,376.248,171.057,45.405,158.756
C05257=1031.267,293.759,376.280,171.053,45.404,158.756
C05258=1031.260,293.511,376.313,171.049,45.405,158.755
C05259=1031.253,293.263,376.345,171.044,45.404,158.755
C05260=1031.246,293.016,376.377,171.040,45.405,158.755
C05261=1031.240,292.768,376.410,171.035,45.405,158.754
C05262=1031.229,292.385,376.459,171.030,45.404,158.753
C05263=1031.219,292.003,376.509,171.023,45.405,158.753
C05264=1031.208,291.620,376.558,171.016,45.405,158.752
C05265=1031.198,291.237,376.608,171.010,45.405,158.751
C05266=1031.191,290.989,376.639,171.006,45.405,158.751
C05267=1031.183,290.741,376.672,171.002,45.405,158.751
C05268=1031.176,290.493,376.703,170.998,45.405,158.750
C05269=1031.170,290.246,376.736,170.993,45.405,158.750
C05270=1031.163,289.998,376.767,170.989,45.406,158.749
C05271=1031.156,289.751,376.800,170.985,45.405,158.749
C05272=1031.149,289.502,376.831,170.981,45.405,158.749
C05273=1031.142,289.254,376.863,170.977,45.406,158.748
C05274=1031.136,289.006,376.896,170.973,45.406,158.748
C05275=1031.129,288.759,376.927,170.969,45.405,158.747
C05276=1031.122,288.511,376.959,170.965,45.406,158.747
C05277=1031.116,288.263,376.991,170.960,45.406,158.746
C05278=1031.109,288.015,377.022,170.956,45.406,158.746
C05279=1031.102,287.767,377.054,170.953,45.406,158.746
C05280=1031.095,287.519,377.087,170.948,45.406,158.745
C05281=1031.089,287.271,377.118,170.944,45.406,158.745
C05282=1031.082,287.023,377.149,170.940,45.407,158.744
C05283=1031.075,286.776,377.182,170.936,45.407,158.744
C05284=1031.068,286.528,377.213,170.932,45.407,158.744
C05285=1031.061,286.280,377.244,170.927,45.407,158.743
C05286=1031.055,286.032,377.276,170.924,45.407,158.743
C05287=1031.048,285.785,377.307,170.920,45.407,158.742
C05288=1031.041,285.537,377.339,170.916,45.407,158.742
C05289=1031.034,285.289,377.370,170.911,45.408,158.742
C05290=1031.027,285.041,377.403,170.908,45.408,158.741
C05291=1031.020,284.793,377.434,170.904,45.408,158.741
C05292=1031.013,284.545,377.465,170.899,45.408,158.741
C05293=1031.007,284.297,377.497,170.896,45.409,158.740
C05294=1031.000,284.049,377.528,170.892,45.409,158.740
C05295=1030.993,283.801,377.560,170.887,45.409,158.739
C05296=1030.986,283.553,377.591,170.884,45.409,158.739
C05297=1030.980,283.305,377.623,170.880,45.410,158.739
C05298=1030.972,283.058,377.653,170.875,45.410,158.738
C05299=1030.966,282.810,377.685,170.871,45.410,158.738
C05300=1030.959,282.562,377.716,170.868,45.410,158.738
C05301=1030.952,282.314,377.747,170.864,45.411,158.737
C05302=1030.946,282.066,377.779,170.859,45.411,158.737
C05303=1030.939,281.818,377.810,170.856,45.411,158.737
C05304=1030.932,281.570,377.841,170.852,45.411,158.736
C05305=1030.925,281.322,377.873,170.847,45.412,158.736
C05306=1030.919,281.074,377.904,170.844,45.412,158.736
C05307=1030.912,280.826,377.936,170.840,45.413,158.735
C05308=1030.905,280.578,377.967,170.837,45.413,158.735
C05309=1030.899,280.330,377.998,170.832,45.413,158.735
C05310=1030.891,280.082,378.029,170.828,45.413,158.734
C05311=1030.885,279.834,378.060,170.825,45.413,158.734
C05312=1030.879,279.587,378.091,170.821,45.414,158.733
C05313=1030.872,279.339,378.123,170.816,45.414,158.733
C05314=1030.865,279.091,378.153,170.813,45.414,158.733
C05315=1030.859,278.843,378.185,170.809,45.415,158.732
C05316=1030.852,278.595,378.216,170.806,45.415,158.732
C05317=1030.845,278.347,378.248,170.801,45.415,158.732
C05318=1030.835,277.976,378.293,170.796,45.416,158.731
C05319=1030.825,277.605,378.340,170.789,45.416,158.731
C05320=1030.815,277.235,378.386,170.784,45.417,158.730
C05321=1030.805,276.864,378.432,170.778,45.417,158.730
C05322=1030.798,276.616,378.463,170.775,45.418,158.730
C05323=1030.791,276.368,378.494,170.770,45.418,158.729
C05324=1030.784,276.120,378.525,170.766,45.419,158.729
C05325=1030.779,275.872,378.555,170.763,45.419,158.728
C05326=1030.771,275.625,378.586,170.759,45.420,158.728
C05327=1030.765,275.376,378.617,170.755,45.420,158.728
C05328=1030.758,275.128,378.648,170.751,45.420,158.728
C05329=1030.751,274.880,378.678,170.747,45.421,158.727
C05330=1030.744,274.632,378.710,170.744,45.421,158.727
C05331=1030.738,274.385,378.740,170.739,45.421,158.727
C05332=1030.731,274.136,378.770,170.736,45.422,158.726
C05333=1030.724,273.888,378.802,170.732,45.422,158.726
C05334=1030.718,273.640,378.832,170.729,45.422,158.726
C05335=1030.710,273.392,378.863,170.725,45.423,158.725
C05336=1030.705,273.144,378.894,170.720,45.424,158.725
C05337=1030.697,272.896,378.924,170.717,45.424,158.725
C05338=1030.691,272.648,378.955,170.713,45.425,158.725
C05339=1030.684,272.400,378.985,170.710,45.425,158.724
C05340=1030.678,272.152,379.016,170.706,45.426,158.724
C05341=1030.671,271.904,379.047,170.702,45.426,158.724
C05342=1030.664,271.656,379.077,170.698,45.427,158.723
C05343=1030.657,271.408,379.108,170.694,45.427,158.723
C05344=1030.651,271.160,379.138,170.691,45.428,158.723
C05345=1030.644,270.912,379.169,170.687,45.428,158.723
C05346=1030.637,270.664,379.199,170.684,45.429,158.722
C05347=1030.631,270.416,379.230,170.679,45.429,158.722
C05348=1030.624,270.168,379.260,170.676,45.430,158.722
C05349=1030.618,269.919,379.290,170.672,45.430,158.721
C05350=1030.610,269.671,379.321,170.669,45.431,158.721
C05351=1030.604,269.424,379.351,170.665,45.431,158.721
C05352=1030.597,269.176,379.382,170.661,45.432,158.721
C05353=1030.590,268.928,379.412,170.657,45.432,158.720
C05354=1030.584,268.680,379.442,170.653,45.433,158.720
C05355=1030.577,268.432,379.472,170.650,45.434,158.720
C05356=1030.570,268.183,379.503,170.646,45.434,158.720
C05357=1030.564,267.936,379.533,170.643,45.435,158.719
C05358=1030.557,267.687,379.563,170.639,45.435,158.719
C05359=1030.551,267.439,379.594,170.636,45.436,158.719
C05360=1030.544,267.191,379.623,170.632,45.437,158.719
C05361=1030.537,266.943,379.654,170.628,45.437,158.718
C05362=1030.530,266.695,379.684,170.624,45.438,158.718
C05363=1030.524,266.447,379.714,170.621,45.438,158.718
C05364=1030.517,266.199,379.744,170.617,45.439,158.717
C05365=1030.510,265.951,379.774,170.614,45.439,158.717
C05366=1030.504,265.703,379.805,170.610,45.440,158.717
C05367=1030.497,265.454,379.834,170.607,45.440,158.717
C05368=1030.490,265.206,379.864,170.603,45.441,158.717
C05369=1030.483,264.958,379.894,170.599,45.442,158.716
C05370=1030.477,264.710,379.924,170.595,45.442,158.716
C05371=1030.470,264.462,379.954,170.592,45.443,158.716
C05372=1030.463,264.214,379.985,170.588,45.444,158.716
C05373=1030.457,263.966,380.014,170.585,45.444,158.715
C05374=1030.447,263.599,380.058,170.579,45.445,158.715
C05375=1030.437,263.234,380.102,170.574,45.447,158.715
C05376=1030.427,262.868,380.146,170.568,45.447,158.714
C05377=1030.418,262.502,380.191,170.563,45.448,158.714
C05378=1030.411,262.254,380.221,170.560,45.449,158.714
C05379=1030.404,262.006,380.251,170.556,45.450,158.714
C05380=1030.398,261.757,380.280,170.553,45.450,158.713
C05381=1030.391,261.510,380.310,170.549,45.451,158.713
C05382=1030.385,261.261,380.340,170.546,45.452,158.713
C05383=1030.378,261.013,380.369,170.542,45.453,158.713
C05384=1030.370,260.765,380.399,170.539,45.453,158.712
C05385=1030.364,260.517,380.428,170.535,45.454,158.712
C05386=1030.357,260.269,380.458,170.532,45.455,158.712
C05387=1030.351,260.021,380.487,170.528,45.456,158.712
C05388=1030.344,259.773,380.517,170.525,45.457,158.712
C05389=1030.337,259.524,380.547,170.521,45.457,158.711
C05390=1030.330,259.277,380.576,170.518,45.458,158.711
C05391=1030.323,259.028,380.605,170.513,45.459,158.711
C05392=1030.316,258.780,380.634,170.510,45.460,158.711
C05393=1030.309,258.531,380.664,170.506,45.461,158.711
C05394=1030.303,258.283,380.693,170.503,45.461,158.710
C05395=1030.295,258.035,380.723,170.499,45.462,158.710
C05396=1030.289,257.787,380.752,170.496,45.463,158.710
C05397=1030.282,257.538,380.781,170.492,45.464,158.710
C05398=1030.275,257.291,380.811,170.489,45.465,158.710
C05399=1030.269,257.042,380.841,170.485,45.466,158.709
C05400=1030.262,256.794,380.870,170.482,45.466,158.709
C05401=1030.255,256.547,380.899,170.478,45.467,158.709
C05402=1030.248,256.298,380.928,170.475,45.468,158.709
C05403=1030.242,256.050,380.957,170.471,45.469,158.709
C05404=1030.235,255.802,380.987,170.468,45.470,158.709
C05405=1030.229,255.553,381.016,170.465,45.470,158.708
C05406=1030.221,255.305,381.045,170.461,45.471,158.708
C05407=1030.215,255.057,381.074,170.458,45.472,158.708
C05408=1030.208,254.809,381.104,170.454,45.473,158.708
C05409=1030.201,254.560,381.133,170.451,45.474,158.708
C05410=1030.195,254.312,381.162,170.447,45.475,158.708
C05411=1030.187,254.064,381.191,170.444,45.476,158.707
C05412=1030.181,253.816,381.220,170.440,45.477,158.707
C05413=1030.175,253.568,381.250,170.437,45.478,158.707
C05414=1030.168,253.319,381.279,170.434,45.478,158.707
C05415=1030.162,253.071,381.309,170.430,45.479,158.707
C05416=1030.155,252.823,381.337,170.427,45.480,158.706
C05417=1030.148,252.575,381.366,170.423,45.481,158.706
C05418=1030.141,252.326,381.395,170.420,45.482,158.706
C05419=1030.135,252.078,381.424,170.417,45.483,158.706
C05420=1030.128,251.830,381.455,170.413,45.484,158.706
C05421=1030.121,251.582,381.483,170.410,45.484,158.706
C05422=1030.115,251.334,381.512,170.406,45.485,158.705
C05423=1030.108,251.085,381.541,170.403,45.486,158.705
C05424=1030.102,250.837,381.571,170.400,45.487,158.705
C05425=1030.095,250.589,381.600,170.396,45.488,158.705
C05426=1030.088,250.341,381.628,170.393,45.489,158.705
C05427=1030.082,250.092,381.657,170.389,45.490,158.705
C05428=1030.075,249.844,381.686,170.386,45.491,158.704
C05429=1030.069,249.596,381.716,170.383,45.491,158.704
C05430=1030.059,249.229,381.758,170.378,45.493,158.704
C05431=1030.049,248.861,381.801,170.373,45.494,158.704
C05432=1030.040,248.494,381.845,170.368,45.496,158.704
C05433=1030.030,248.127,381.887,170.363,45.497,158.703
C05434=1030.024,247.879,381.916,170.360,45.497,158.703
C05435=1030.017,247.629,381.945,170.356,45.499,158.703
C05436=1030.010,247.382,381.973,170.353,45.500,158.703
C05437=1030.004,247.134,382.002,170.350,45.500,158.703
C05438=1029.998,246.885,382.031,170.346,45.501,158.702
C05439=1029.991,246.637,382.060,170.343,45.503,158.702
C05440=1029.985,246.388,382.090,170.340,45.503,158.702
C05441=1029.978,246.141,382.118,170.336,45.504,158.702
C05442=1029.971,245.892,382.147,170.333,45.505,158.702
C05443=1029.965,245.644,382.176,170.330,45.506,158.702
C05444=1029.959,245.396,382.205,170.326,45.507,158.702
C05445=1029.952,245.148,382.233,170.323,45.508,158.702
C05446=1029.945,244.899,382.263,170.320,45.509,158.701
C05447=1029.939,244.651,382.292,170.316,45.510,158.701
C05448=1029.933,244.403,382.321,170.313,45.511,158.701
C05449=1029.926,244.154,382.348,170.310,45.512,158.701
C05450=1029.920,243.906,382.377,170.306,45.513,158.701
C05451=1029.913,243.658,382.406,170.303,45.514,158.701
C05452=1029.907,243.410,382.434,170.300,45.515,158.701
C05453=1029.899,243.161,382.463,170.297,45.516,158.700
C05454=1029.893,242.913,382.492,170.294,45.517,158.700
C05455=1029.886,242.664,382.520,170.291,45.518,158.700
